# B&R Automation Studio project TrakBasisProject
Automation Studio 6.7.0.187; technology packages: mappCockpit 6.7.0, mappMotion 6.7.2, mappView 6.7.0, OpcUaCs 6.7.0

## Configuration Config1

CPU 5PC900.TS17-00, AutomationRuntime 6.7.8, Build 11.3.0

### Task classes (Cpu.sw)
```
Cyclic#1 (cycle 800 us, tolerance 0 us):
  TrakCtrl <- TrakBasis.TrakCtrl.prg
  utTrakCtrl <- UnitTest.utTrakCtrl.utTrakCtrl.prg
Cyclic#8 (cycle 9600 us):
  TrakHmiCtr <- TrakHmi.TrakHmiCtrl.prg
DataObjects: McAcpSys
NcDataObjects: McDriveLog
Binaries: FWRules, TCData, udbdef, mvLoader, mvConfig, McAcpSim, McAcpDrv, User, iomap, Config_1, arconfig, asfw, ashwac, sysconf, Settings, Role, UaCsConfig, ashwd, Config_3, mCoWebSc, Config_2, BRRole, Hierarchy, TrakHmi
Libraries: runtime, AsZip, FileIO, AsIODiag, AsBrStr, standard, AsARCfg, sys_lib, UnitTest, UtMgr, UtWs, McBase, MpBase, MpAxis, McAcpAx, McAcpTrak, McAxis, CoTrace, arsvcreg, astime, arssl, uacoalprv, powerlnk, AsIecCon, UaCoal, AsEPL, AsIOAcc, AsIoTrc, UaCore, arcoal
```

### Hardware
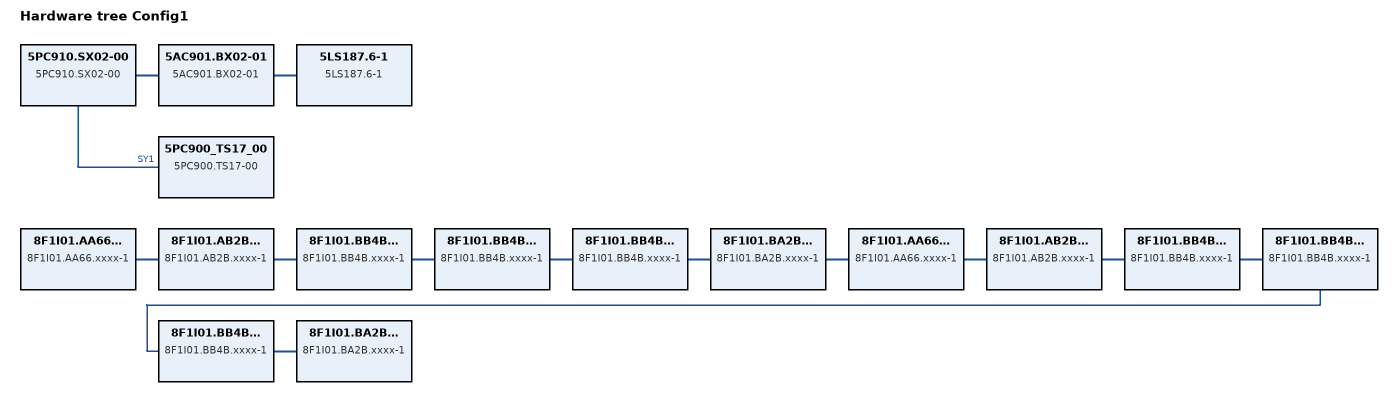
```
5AC901.BX02-01 : 5AC901.BX02-01 v1.1.1.0  [SY -> 5PC910.SX02-00.SY3]
5LS187.6-1 : 5LS187.6-1 v1.10.0.0  [SL -> 5AC901.BX02-01.SL2]
  Connector IF2:
    CycleTime = 800
    EplNatSubnet = 192.168.102.0
5PC900_TS17_00 : 5PC900.TS17-00 v2.2.0.0  [SY -> 5PC910.SX02-00.SY1]
  ConfigurationID = TrakBasisProject_Config1
  UserPartitionSize = 200
  Simulation = 1
  RemMemDevice = PCI.2.LS187.SRAM
  RemMemSize = 20000
  RemanentGlobalPvSize = 3000
  MotionLoggerSize = 2048000
  TimerDeviceType = EPLX2X
  TimerDevice = 5LS187.6-1.IF2
  IdleTaskClass = 3
  TaskClassIdleTime = 1600
  Cyclic1Duration = 800
  Cyclic1Tolerance = 0
  Cyclic1Stack = 256000
  Cyclic1Output = 1
  Cyclic2Duration = 1600
  Cyclic2Tolerance = 1600
  Cyclic3Duration = 20000
  Cyclic3Tolerance = 40000
  Cyclic8Duration = 9600
  Cyclic8Stack = 100000
  FileDevice1
  FileDeviceName1 = SvgData
  FileDevicePath1 = USER_PATH
  ActivateFtpServer = 1
  FtpUser1
  FtpUsername1 = BR
  FtpUserPassword1 = sCAcS4M0KXkF12D2Ev+1iYDIV5DbZPUJhKJtxWH0zr0=  // BR
  FtpUserSalt1 = M7Jis0HY
  FTPAccessRight1 = 0
  FTPdevice1 = ALL
  ActivateWebServer = 1
  WebServerProtocol = 1
  ActivateSdm = 1
5PC910.SX02-00 : 5PC910.SX02-00 v2.1.2.0
  Connector IF1:
    AssignedOperatingSystem = ARemb
  Connector IF3:
    AssignedOperatingSystem = ARemb
    ActivateDevice = 1
  Connector IF4:
    AssignedOperatingSystem = ARemb
    ActivateDevice = 1
    ActivateSnmp = 2
  Connector IF5:
    AssignedOperatingSystem = ARemb
  Connector IF6:
    AssignedOperatingSystem = ARemb
  Connector IF7:
    AssignedOperatingSystem = ARemb
  Connector IF8:
    AssignedOperatingSystem = ARemb
  Connector IF9:
    AssignedOperatingSystem = ARemb
8F1I01.AA66.xxxx-1 : 8F1I01.AA66.xxxx-1 v1.0.1.0 (NodeNumber=12)  [PLK2 -> 8F1I01.AB2B.xxxx-1.PLK1 [Cable Type=PowerlinkCable, Length=10, Version=1.0.0.3]]
  DriveConfiguration:
    McTypeID = LLMConfig
  DriveConfiguration/Segment:
    Shape = STRAIGHT660
    SegmentReference = Seg_7
    SegmentSectorDirection = Positive
  DriveConfiguration/Segment/Compensation:
    ElongationCompensation = UseAssemblySetting
    ACC = Inactive
  DriveConfiguration/Segment:
    StopReaction = UseAssemblySetting
    SpeedFilter = UseAssemblySetting
    PositionControllerLagMonitor = UseAssemblySetting
8F1I01.AA66.xxxx-1a : 8F1I01.AA66.xxxx-1 v1.0.1.0 (NodeNumber=1)  [PLK1 -> 8F1I01.BA2B.xxxx-1a.PLK2 [Cable Type=PowerlinkCable, Length=10, Version=1.0.0.3]; PLK2 -> 8F1I01.AB2B.xxxx-1a.PLK1 [Cable Type=PowerlinkCable, Length=10, Version=1.0.0.3]; PLK3 -> 5LS187.6-1.IF2 [Cable Type=PowerlinkCable, Length=10, Version=1.0.0.3]]
  DriveConfiguration:
    McTypeID = LLMConfig
  DriveConfiguration/Segment:
    Shape = STRAIGHT660
    SegmentReference = Seg_1
    SegmentSectorDirection = Positive
  DriveConfiguration/Segment/Compensation:
    ElongationCompensation = UseAssemblySetting
    ACC = Inactive
  DriveConfiguration/Segment:
    StopReaction = UseAssemblySetting
    SpeedFilter = UseAssemblySetting
    PositionControllerLagMonitor = UseAssemblySetting
8F1I01.AB2B.xxxx-1 : 8F1I01.AB2B.xxxx-1 v1.0.1.0 (NodeNumber=11)  [PLK1 -> 8F1I01.AA66.xxxx-1.PLK2 [Cable Type=PowerlinkCable, Length=10, Version=1.0.0.3]; PLK2 -> 8F1I01.BB4B.xxxx-1c.PLK1 [Cable Type=PowerlinkCable, Length=10, Version=1.0.0.3]]
  DriveConfiguration:
    McTypeID = LLMConfig
  DriveConfiguration/Segment:
    Shape = STRAIGHT105_TO_CIRCULAR
    SegmentReference = Seg_8
    SegmentSectorDirection = Positive
  DriveConfiguration/Segment/Compensation:
    ElongationCompensation = UseAssemblySetting
    ACC = Inactive
  DriveConfiguration/Segment:
    StopReaction = UseAssemblySetting
    SpeedFilter = UseAssemblySetting
    PositionControllerLagMonitor = UseAssemblySetting
8F1I01.AB2B.xxxx-1a : 8F1I01.AB2B.xxxx-1 v1.0.1.0 (NodeNumber=2)  [PLK1 -> 8F1I01.AA66.xxxx-1a.PLK2 [Cable Type=PowerlinkCable, Length=10, Version=1.0.0.3]; PLK2 -> 8F1I01.BB4B.xxxx-1.PLK1 [Cable Type=PowerlinkCable, Length=10, Version=1.0.0.3]]
  DriveConfiguration:
    McTypeID = LLMConfig
  DriveConfiguration/Segment:
    Shape = STRAIGHT105_TO_CIRCULAR
    SegmentReference = Seg_2
    SegmentSectorDirection = Positive
  DriveConfiguration/Segment/Compensation:
    ElongationCompensation = UseAssemblySetting
    ACC = Inactive
  DriveConfiguration/Segment:
    StopReaction = UseAssemblySetting
    SpeedFilter = UseAssemblySetting
    PositionControllerLagMonitor = UseAssemblySetting
8F1I01.BA2B.xxxx-1 : 8F1I01.BA2B.xxxx-1 v1.0.1.0 (NodeNumber=7)  [PLK1 -> 8F1I01.BB4B.xxxx-1b.PLK2 [Cable Type=PowerlinkCable, Length=10, Version=1.0.0.3]]
  DriveConfiguration:
    McTypeID = LLMConfig
  DriveConfiguration/Segment:
    Shape = CIRCULAR_TO_STRAIGHT105
    SegmentReference = Seg_6
    SegmentSectorDirection = Positive
  DriveConfiguration/Segment/Compensation:
    ElongationCompensation = UseAssemblySetting
    ACC = Inactive
  DriveConfiguration/Segment:
    StopReaction = UseAssemblySetting
    SpeedFilter = UseAssemblySetting
    PositionControllerLagMonitor = UseAssemblySetting
8F1I01.BA2B.xxxx-1a : 8F1I01.BA2B.xxxx-1 v1.0.1.0  [PLK1 -> 8F1I01.BB4B.xxxx-1e.PLK2 [Cable Type=PowerlinkCable, Length=10, Version=1.0.0.3]; PLK2 -> 8F1I01.AA66.xxxx-1a.PLK1 [Cable Type=PowerlinkCable, Length=10, Version=1.0.0.3]]
  DriveConfiguration:
    McTypeID = LLMConfig
  DriveConfiguration/Segment:
    Shape = CIRCULAR_TO_STRAIGHT105
    SegmentReference = Seg_12
    SegmentSectorDirection = Positive
  DriveConfiguration/Segment/Compensation:
    ElongationCompensation = UseAssemblySetting
    ACC = Inactive
  DriveConfiguration/Segment:
    StopReaction = UseAssemblySetting
    SpeedFilter = UseAssemblySetting
    PositionControllerLagMonitor = UseAssemblySetting
8F1I01.BB4B.xxxx-1 : 8F1I01.BB4B.xxxx-1 v1.0.1.0 (NodeNumber=4)  [PLK1 -> 8F1I01.AB2B.xxxx-1a.PLK2 [Cable Type=PowerlinkCable, Length=10, Version=1.0.0.3]; PLK2 -> 8F1I01.BB4B.xxxx-1a.PLK1 [Cable Type=PowerlinkCable, Length=10, Version=1.0.0.3]]
  DriveConfiguration:
    McTypeID = LLMConfig
  DriveConfiguration/Segment:
    Shape = CIRCULAR
    SegmentReference = Seg_3
    SegmentSectorDirection = Positive
  DriveConfiguration/Segment/Compensation:
    ElongationCompensation = UseAssemblySetting
    ACC = Inactive
  DriveConfiguration/Segment:
    StopReaction = UseAssemblySetting
    SpeedFilter = UseAssemblySetting
    PositionControllerLagMonitor = UseAssemblySetting
8F1I01.BB4B.xxxx-1a : 8F1I01.BB4B.xxxx-1 v1.0.1.0 (NodeNumber=5)  [PLK1 -> 8F1I01.BB4B.xxxx-1.PLK2 [Cable Type=PowerlinkCable, Length=10, Version=1.0.0.3]; PLK2 -> 8F1I01.BB4B.xxxx-1b.PLK1 [Cable Type=PowerlinkCable, Length=10, Version=1.0.0.3]]
  DriveConfiguration:
    McTypeID = LLMConfig
  DriveConfiguration/Segment:
    Shape = CIRCULAR
    SegmentReference = Seg_4
    SegmentSectorDirection = Positive
  DriveConfiguration/Segment/Compensation:
    ElongationCompensation = UseAssemblySetting
    ACC = Inactive
  DriveConfiguration/Segment:
    StopReaction = UseAssemblySetting
    SpeedFilter = UseAssemblySetting
    PositionControllerLagMonitor = UseAssemblySetting
8F1I01.BB4B.xxxx-1b : 8F1I01.BB4B.xxxx-1 v1.0.1.0 (NodeNumber=6)  [PLK1 -> 8F1I01.BB4B.xxxx-1a.PLK2 [Cable Type=PowerlinkCable, Length=10, Version=1.0.0.3]; PLK2 -> 8F1I01.BA2B.xxxx-1.PLK1 [Cable Type=PowerlinkCable, Length=10, Version=1.0.0.3]]
  DriveConfiguration:
    McTypeID = LLMConfig
  DriveConfiguration/Segment:
    Shape = CIRCULAR
    SegmentReference = Seg_5
    SegmentSectorDirection = Positive
  DriveConfiguration/Segment/Compensation:
    ElongationCompensation = UseAssemblySetting
    ACC = Inactive
  DriveConfiguration/Segment:
    StopReaction = UseAssemblySetting
    SpeedFilter = UseAssemblySetting
    PositionControllerLagMonitor = UseAssemblySetting
8F1I01.BB4B.xxxx-1c : 8F1I01.BB4B.xxxx-1 v1.0.1.0 (NodeNumber=10)  [PLK1 -> 8F1I01.AB2B.xxxx-1.PLK2 [Cable Type=PowerlinkCable, Length=10, Version=1.0.0.3]; PLK2 -> 8F1I01.BB4B.xxxx-1d.PLK1 [Cable Type=PowerlinkCable, Length=10, Version=1.0.0.3]]
  DriveConfiguration:
    McTypeID = LLMConfig
  DriveConfiguration/Segment:
    Shape = CIRCULAR
    SegmentReference = Seg_9
    SegmentSectorDirection = Positive
  DriveConfiguration/Segment/Compensation:
    ElongationCompensation = UseAssemblySetting
    ACC = Inactive
  DriveConfiguration/Segment:
    StopReaction = UseAssemblySetting
    SpeedFilter = UseAssemblySetting
    PositionControllerLagMonitor = UseAssemblySetting
8F1I01.BB4B.xxxx-1d : 8F1I01.BB4B.xxxx-1 v1.0.1.0 (NodeNumber=9)  [PLK1 -> 8F1I01.BB4B.xxxx-1c.PLK2 [Cable Type=PowerlinkCable, Length=10, Version=1.0.0.3]; PLK2 -> 8F1I01.BB4B.xxxx-1e.PLK1 [Cable Type=PowerlinkCable, Length=10, Version=1.0.0.3]]
  DriveConfiguration:
    McTypeID = LLMConfig
  DriveConfiguration/Segment:
    Shape = CIRCULAR
    SegmentReference = Seg_10
    SegmentSectorDirection = Positive
  DriveConfiguration/Segment/Compensation:
    ElongationCompensation = UseAssemblySetting
    ACC = Inactive
  DriveConfiguration/Segment:
    StopReaction = UseAssemblySetting
    SpeedFilter = UseAssemblySetting
    PositionControllerLagMonitor = UseAssemblySetting
8F1I01.BB4B.xxxx-1e : 8F1I01.BB4B.xxxx-1 v1.0.1.0  [PLK1 -> 8F1I01.BB4B.xxxx-1d.PLK2 [Cable Type=PowerlinkCable, Length=10, Version=1.0.0.3]; PLK2 -> 8F1I01.BA2B.xxxx-1a.PLK1 [Cable Type=PowerlinkCable, Length=10, Version=1.0.0.3]]
  DriveConfiguration:
    McTypeID = LLMConfig
  DriveConfiguration/Segment:
    Shape = CIRCULAR
    SegmentReference = Seg_11
    SegmentSectorDirection = Positive
  DriveConfiguration/Segment/Compensation:
    ElongationCompensation = UseAssemblySetting
    ACC = Inactive
  DriveConfiguration/Segment:
    StopReaction = UseAssemblySetting
    SpeedFilter = UseAssemblySetting
    PositionControllerLagMonitor = UseAssemblySetting
```

### Config_1.assembly - 5PC900_TS17_00/mappMotion/Config_1.assembly
```
Element gAssembly_1 (Type=assembly)
  Tracks:
    Track[1]:
      Segments:
        SegmentRef[1] = ::Seg_1
        SegmentRef[2] = ::Seg_2
        SegmentRef[3] = ::Seg_3
        SegmentRef[4] = ::Seg_4
        SegmentRef[5] = ::Seg_5
        SegmentRef[6] = ::Seg_6
        SegmentRef[7] = ::Seg_7
        SegmentRef[8] = ::Seg_8
        SegmentRef[9] = ::Seg_9
        SegmentRef[10] = ::Seg_10
        SegmentRef[11] = ::Seg_11
        SegmentRef[12] = ::Seg_12
  CommonSegmentSettings:
    ControllerParameters:
      DefaultParameter:
        Controller:
          Position:
            ProportionalGain = 150
          Speed:
            ProportionalGain = 120
          FeedForward:
            TotalMass = 1.25
            ForcePositive = 1.0
            ForceNegative = 1.0
  Shuttles:
    MaxShuttleCount = 40
    ShuttleStereotypes:
      ShuttleStRef[1] = ShuttleStereotype_1
    MagnetPlateConfigurations:
      ShuttleType[1] = 8F1Sx.102.xxxxxx-x
    BackupShuttleData = Used
      BackupVar = ::gTrakShBackupRestoreData
```

### Config_2.sector - 5PC900_TS17_00/mappMotion/Config_2.sector
```
Element Sector_1 (Type=sector)
  Type:
    StartSegment:
      SegmentRef = ::Seg_1
    IntermediateSegments:
      SegmentRef[1] = ::Seg_2
      SegmentRef[2] = ::Seg_3
      SegmentRef[3] = ::Seg_4
      SegmentRef[4] = ::Seg_5
      SegmentRef[5] = ::Seg_6
      SegmentRef[6] = ::Seg_7
      SegmentRef[7] = ::Seg_8
      SegmentRef[8] = ::Seg_9
      SegmentRef[9] = ::Seg_10
      SegmentRef[10] = ::Seg_11
    EndSegment:
      SegmentRef = ::Seg_12
      PositionRelativeTo = FromEnd
```

### Config_3.shuttlestereotype - 5PC900_TS17_00/mappMotion/Config_3.shuttlestereotype
```
Element ShuttleStereotype_1 (Type=shuttlestereotype)
  MovementLimits:
    Velocity:
      Velocity = 5.5
    Acceleration:
      Acceleration = 40.0
    Deceleration:
      Deceleration = 40.0
```

### Config_4.assemblyfeature - 5PC900_TS17_00/mappMotion/Config_4.assemblyfeature
```
Element Feature_Shuttle_Auto_Attatch (Type=assemblyfeature)
  Type = ShtSectorAutoAttach
    Priority[1]:
      SectorRef = Sector_1
```

## Logical view

Binary libraries used (declarations not repeated): operator, runtime, AsIecCon, astime, AsZip, FileIO, AsIODiag, AsBrStr, standard, McBase 6.3.0, MpBase 6.7.0, MpAxis 6.3.0, McAcpAx 6.3.0, McAcpTrak 6.7.2, McAxis 6.3.0, CoTrace 6.1.0, UtMgr 6.3.0, sys_lib, AsARCfg, UtWs 6.3.0

### Package Logical/Libraries - Global libraries

### TrakBasis.typ
```iecst
(********************************************************************
 * COPYRIGHT - B&R Spain
 ********************************************************************
 * Package: TrakBasis
 * File: TrakBasis.typ
 * Author: B&R Spain
 * Created: July 22, 2024
 * Modified: July 22, 2024
 ********************************************************************
 * Data types of package TrakBasis for mapp Motion
 ********************************************************************)
(*********************************************************************
* TrakCtrl structures
*********************************************************************)

TYPE
	TrakApplicationErrorEnum :
		(
		TRAK_APP_ERROR_NONE := 0,
		TRAK_APP_ERR_SIM_SH_COUNT_MAX := 100,
		TRAK_APP_ERR_SH_COUNT_MAX := 101,
		TRAK_APP_ERR_SEG_COUNT_MAX := 102,
		TRAK_APP_ERR_SEG_INDEX_MAX := 103,
		TRAK_APP_ERR_NO_SEGMENTS := 104
		);
	TrakCtrlType : 	STRUCT  (*Control structure*)
		Command : TrakCtrlCmdType; (*Command structure*)
		Parameter : TrakCtrlParType; (*Parameter structure*)
		Status : TrakCtrlStatusType; (*Status structure*)
	END_STRUCT;
	TrakCtrlCmdType : 	STRUCT  (*Command structure*)
		Power : BOOL; (*Switch on the controller*)
		Move : TrakCtrlCmdMoveType; (*Movement structures*)
		ErrorReset : BOOL; (*Reset the error in assembly*)
		Recover : TrakCtrlCmdRecoverType; (*Shuttle identity recovery commands*)
	END_STRUCT;
	TrakCtrlCmdMoveType : 	STRUCT  (*Movement structures*)
		Absolute : BOOL; (*Elastic move absolute of all the shuttles to a predefined position*)
		Velocity : BOOL; (*Velocity move of all the shuttles within the predefined sector*)
		Halt : BOOL; (*Stops all shuttle movements*)
	END_STRUCT;
	TrakCtrlCmdRecoverType : 	STRUCT  (*Shuttle identity recovery commands*)
		Index : UINT; (*Index in Status.Shuttle[] of the shuttle to identify*)
		UserID : STRING[32]; (*UserID supplied externally (e.g. by a camera recognition system)*)
		Execute : BOOL; (*Assigns UserID to the shuttle at Index*)
		ResetShuttleData : BOOL; (*Wipes the remanent shuttle backup/restore store (mcACPTRAK_RESTORE_RESET_DATA)*)
	END_STRUCT;
	TrakCtrlParType : 	STRUCT  (*Parameter structure*)
		Position : LREAL; (*Position of the commanded movement for the selecred shuttle*)
		Direction : McDirectionEnum; (*Direction of the commanded movement for the selecred shuttle*)
		Speed : REAL; (*Velocity of the commanded movement for the selecred shuttle*)
		Acceleration : REAL; (*Acceleration of the commanded movement for the selecred shuttle*)
		Deceleration : REAL; (*Deceleration of the commanded movement for the selecred shuttle*)
		RestoreEnabled : BOOL; (*The system try to restore shuttle positions after power on*)
		RestoreTolerance : LREAL; (*Discrepancy allowed when restoring position*)
		SimulationParameters : TrakCtrlParSimType; (*Simulation parameter for the trak system*)
	END_STRUCT;
	TrakCtrlParSimType : 	STRUCT  (*Parameter for when trak is being simulated*)
		Position : LREAL; (*Position of first shuttle*)
		Separation : LREAL; (*Separation between shuttles*)
		Quantity : UINT; (*Quantity of the shuttles*)
	END_STRUCT;
	TrakCtrlStatusType : 	STRUCT  (*Status structure*)
		CommunicationReady : BOOL; (*Communication is posible with the assembly*)
		ReadyForPowerOn : BOOL; (*Assembly can be powered on*)
		PowerOn : BOOL; (*Assembly is powered in*)
		MovementDetected : BOOL; (*There are movements in the assembly*)
		Error : BOOL; (*A hardware or application error is active*)
		ErrorInfo : TrakCtrlStatusErrorInfoType; (*Hardware or application error information*)
		AutomaticRestoreSuccess : BOOL; (*TRUE if the automatic restore matched all detected shuttles; FALSE otherwise (some need Command.Recover)*)
		PLCopenState : TrakCtrlStatusPLCopenStateType; (*PLC Open state of the assembly *)
		Segment : ARRAY[0..TRAK_MAX_SEGMENT_MINUS_ONE]OF TrakCtrlStatusSegmentType; (*Overall count of the segments*)
		Shuttle : ARRAY[0..TRAK_MAX_SHUTTLE_MINUS_ONE]OF TrakCtrlStatusShuttleType; (*Overall count of the shuttles*)
	END_STRUCT;
	TrakCtrlStatusErrorInfoType : 	STRUCT  (*Track error related information*)
		ID : DINT; (*The error id of any ocurred error*)
		Text : STRING[255]; (*Error description*)
		Initiator : STRING[32]; (*Error initiator*)
	END_STRUCT;
	TrakCtrlStatusShuttleType : 	STRUCT  (*Overrall numbers of shuttles*)
		Valid : BOOL; (*Shuttle data valid*)
		Axis : McAxisType; (*McAxis of shuttle*)
		ID : UDINT; (*User defined shuttle ID*)
		Name : STRING[32]; (*User defined name identificator*)
		ActSectorType : McAcpTrakSecTypeEnum; (*Shuttle current sector type*)
		ActSector : STRING[32]; (*Shuttle current sector*)
		ActPosition : LREAL; (*Shuttle position on sector*)
		ActVelocity : REAL; (*Shuttle velocity on sector*)
		TotalMoveDistance : LREAL; (*Shuttle total moved distance*)
		IsConvoyMaster : BOOL; (*Shuttle is a convoy master*)
		Pos : McPosType; (*Shuttle position in the coordinate system*)
		State : TrakCtrlStatusShuttleStateType; (*Shuttle state*)
	END_STRUCT;
	TrakCtrlStatusShuttleStateType : 	STRUCT  (*Shuttle PLCopen state*)
		StatusStandStill : BOOL; (*Shuttle is in state Standstill*)
		StatusStopping : BOOL; (*Shuttle is in state Stopping*)
		StatusErrorStop : BOOL; (*Shuttle is in state Errorstop*)
		StatusDiscreteMotion : BOOL; (*Shuttle is in state DiscreteMotion*)
		StatusContinuousMotion : BOOL; (*Shuttle is in state ContinuousMotion*)
		StatusSynchronizedMotion : BOOL; (*Shuttle is in state SynchronizedMotion*)
	END_STRUCT;
	TrakCtrlStatusPLCopenStateType : 	STRUCT  (*PLC Open states of the assembly*)
		Disabled : BOOL; (*Assembly in disabled state*)
		Homing : BOOL; (*Assembly in homing state*)
		Ready : BOOL; (*Assembly in ready state*)
		Stopping : BOOL; (*Assembly in stopping state*)
		ErrorStop : BOOL; (*Assembly in error state*)
		StartUp : BOOL; (*Assembly in start up state*)
		InvalidConfigurartion : BOOL; (*Assembly is invalid*)
	END_STRUCT;
	TrakCtrlStatusSegmentType : 	STRUCT  (*Overrall numbers of segments*)
		Valid : BOOL; (*Segment data valid*)
		Segment : McSegmentType; (*Segment reference*)
		Name : STRING[32]; (*Segment name (used mainly for diagnostics)*)
		State : TrakCtrlStatusSegmentState; (*Segment current PLCopen state*)
		Info : TrakCtrlStatusSegmentInfoType; (*Segment additional information (tempreature, current...etc)*)
	END_STRUCT;
	TrakCtrlStatusSegmentState : 	STRUCT  (*Segment PLCopen state*)
		StatusDisabled : BOOL; (*Segment is in state Disabled*)
		StatusReady : BOOL; (*Segment is in state Ready*)
		StatusErrorStop : BOOL; (*Segment is in state ErrorStop*)
		InvalidConfig : BOOL; (*Segment has an invalid configuration*)
	END_STRUCT;
	TrakCtrlStatusSegmentInfoType : 	STRUCT  (*Additional segment information*)
		TempBalancer : REAL; (*Internal segment temperature*)
		TempSensor : REAL; (*Backside segment temperature*)
		TempAir : REAL; (*CPU segment temperature*)
		Voltage : REAL; (*DC segment voltage*)
		PowerConsumption : REAL; (*Power consumption of the segment*)
	END_STRUCT;
END_TYPE
```

### TrakBasis.var
```iecst
(**)
(********************************************************************
 * CONSTANT VALUE
********************************************************************)
VAR CONSTANT
	TRAK_MAX_SEGMENT : UINT := 12;
	TRAK_MAX_SHUTTLE : UINT := 40; (*Maximum number of shuttles. This value must match the assembly configuration file*)
	TRAK_MAX_SEGMENT_MINUS_ONE : UINT := TRAK_MAX_SEGMENT-1;
	TRAK_MAX_SHUTTLE_MINUS_ONE : UINT := TRAK_MAX_SHUTTLE-1;
	TRAK_SH_USER_DATA_SIZE : UINT := 0; (*Bytes reserved per shuttle in User data size.This value must match the shuttle stereotype configuration file*)
	// Per B&R docs: array size must be at least MaxShuttleCount * (68 + user data size)
	TRAK_SH_BACKUP_SIZE_MINUS_ONE : UINT := (TRAK_MAX_SHUTTLE*(68+TRAK_SH_USER_DATA_SIZE))-1;
END_VAR
(********************************************************************
 * Global control variable
********************************************************************)
VAR
	gTrakCtrl : TrakCtrlType;
END_VAR
(********************************************************************
 * Backup and restore data - referenced by name from the assembly's
 * "Backup and restore data" configuration element (Config_1.assembly)
********************************************************************)
VAR RETAIN
	gTrakShBackupRestoreData : ARRAY[0..TRAK_SH_BACKUP_SIZE_MINUS_ONE] OF USINT;
END_VAR
```

### Program Logical/TrakBasis/TrakCtrl (IEC)

#### Reference.st
```iecst
(********************************************************************
 * COPYRIGHT - B&R Spain
 ********************************************************************
 * Program: TrakCtrl
 * File: References.st
 * Author: B&R Spain
 * Created: July 22, 2024
 * Modified: July 22, 2024
 ********************************************************************
 * Implementation of program TrakCtrl
 ********************************************************************
 * Gets the references to the structures
 ********************************************************************)
ACTION References:

	// Obtain the address of the global assembly structure. This pointer can be used in other places to read/write the assembly's data.
	AdrAssembly := ADR(gAssembly_1);
	// Obtain the address of the default sector structure where initial shuttle movements will be performed.
	AdrSector := ADR(Sector_1);
	// Store the name of the global assembly for identification or logging purposes.
	AssemblyName := 'gAssembly_1';
	// Access the address of gTrakCtrl using the built-in ACCESS operator. This ensures pTrakCtrl points directly to gTrakCtrl for control operations.
	pTrakCtrl ACCESS ADR(gTrakCtrl);

END_ACTION
```

#### InitSequence.st
```iecst
//********************************************************************
// COPYRIGHT - B&R Spain
//********************************************************************
// Program: TrakCtrl
// File: InitSequence.st
// Author: B&R Spain
// Created: July 22, 2024
//********************************************************************
// Implementation of program TrakCtrl
//********************************************************************
// This action implements a state machine to initialize the AcoposTrak system.
//********************************************************************

ACTION InitSequence:

	// State machine controlling the initialization of the AcoposTrak system
	CASE InitState OF

		INIT_STATE_SET_PARAMETER:

			// Set default motion parameters before communicating with the trak
			pTrakCtrl.Parameter.Speed := 0.5;
			pTrakCtrl.Parameter.Acceleration := 5.0;
			pTrakCtrl.Parameter.Deceleration := 5.0;
			pTrakCtrl.Parameter.Position := 0.0;
			pTrakCtrl.Parameter.Direction := mcDIR_POSITIVE;

			// Additional parameters for simulation and restore operations
			pTrakCtrl.Parameter.SimulationParameters.Position := 0.1;
			pTrakCtrl.Parameter.SimulationParameters.Quantity := 20;
			pTrakCtrl.Parameter.SimulationParameters.Separation := 0.06;
			pTrakCtrl.Parameter.RestoreEnabled := TRUE;
			pTrakCtrl.Parameter.RestoreTolerance := 0.25;

			InitState := INIT_STATE_CHECK_ASM_COMM;

		INIT_STATE_CHECK_ASM_COMM:

			 // Verify that the assembly is ready for communication
			IF (MC_BR_AsmReadInfo_AcpTrak_0.AssemblyInfo.CommunicationReady) THEN
				InitState := INIT_STATE_ASM_RDY_TO_POWER;
			END_IF

		INIT_STATE_ASM_RDY_TO_POWER:

			// Verify that the assembly is ready to be powered on
			IF (MC_BR_AsmReadInfo_AcpTrak_0.AssemblyInfo.ReadyForPowerOn) THEN
				InitState := INIT_STATE_GET_SEGMENT;
			END_IF

		INIT_STATE_GET_SEGMENT:

			// Start retrieving segment information
			MC_BR_AsmGetSegment_AcpTrak_0.Enable := TRUE;
			MC_BR_AsmGetSegment_AcpTrak_0.Next := FALSE;
			Counter := 0;

			InitState := INIT_STATE_GET_SEGMENT_WAIT;

		INIT_STATE_GET_SEGMENT_WAIT:

			IF (MC_BR_AsmGetSegment_AcpTrak_0.Error) THEN
				MC_BR_AsmGetSegment_AcpTrak_0.Enable := FALSE;
				InitState := INIT_STATE_ERROR;

			// If there's no error, check if valid data is available
			ELSIF (MC_BR_AsmGetSegment_AcpTrak_0.Valid) THEN

				// Store the total amount of segments
				TotalCountSegment := MC_BR_AsmGetSegment_AcpTrak_0.TotalCount;

				// An assembly without segments cannot be initialized
				IF (TotalCountSegment = 0) THEN
					MC_BR_AsmGetSegment_AcpTrak_0.Enable := FALSE;
					MC_BR_AsmGetSegment_AcpTrak_0.Next := FALSE;
					pTrakCtrl.Status.Error := TRUE;
					pTrakCtrl.Status.ErrorInfo.ID := TRAK_APP_ERR_NO_SEGMENTS;
					pTrakCtrl.Status.ErrorInfo.Initiator := 'Application';
					pTrakCtrl.Status.ErrorInfo.Text := 'No segments detected in the assembly. Initialization aborted.';
					InitState := INIT_STATE_ERROR;

				// The configured array must be able to hold every detected segment
				ELSIF (TotalCountSegment > TRAK_MAX_SEGMENT) THEN
					MC_BR_AsmGetSegment_AcpTrak_0.Enable := FALSE;
					MC_BR_AsmGetSegment_AcpTrak_0.Next := FALSE;
					pTrakCtrl.Status.Error := TRUE;
					pTrakCtrl.Status.ErrorInfo.ID := TRAK_APP_ERR_SEG_COUNT_MAX;
					pTrakCtrl.Status.ErrorInfo.Initiator := 'Application';
					AuxString := UINT_TO_STRING(TotalCountSegment);
					pTrakCtrl.Status.ErrorInfo.Text := CONCAT('Detected segment count (',AuxString);
					pTrakCtrl.Status.ErrorInfo.Text := CONCAT(pTrakCtrl.Status.ErrorInfo.Text,') exceeds TRAK_MAX_SEGMENT limit (');
					AuxString := UINT_TO_STRING(TRAK_MAX_SEGMENT);
					pTrakCtrl.Status.ErrorInfo.Text := CONCAT(pTrakCtrl.Status.ErrorInfo.Text,AuxString);
					pTrakCtrl.Status.ErrorInfo.Text := CONCAT(pTrakCtrl.Status.ErrorInfo.Text,'). Initialization aborted.');
					InitState := INIT_STATE_ERROR;

				// Protect the destination array if the FB returns inconsistent count information
				ELSIF (Counter >= TRAK_MAX_SEGMENT) THEN
					MC_BR_AsmGetSegment_AcpTrak_0.Enable := FALSE;
					MC_BR_AsmGetSegment_AcpTrak_0.Next := FALSE;
					pTrakCtrl.Status.Error := TRUE;
					pTrakCtrl.Status.ErrorInfo.ID := TRAK_APP_ERR_SEG_INDEX_MAX;
					pTrakCtrl.Status.ErrorInfo.Initiator := 'Application';
					AuxString := UINT_TO_STRING(Counter);
					pTrakCtrl.Status.ErrorInfo.Text := CONCAT('Segment index (',AuxString);
					pTrakCtrl.Status.ErrorInfo.Text := CONCAT(pTrakCtrl.Status.ErrorInfo.Text,') is outside TRAK_MAX_SEGMENT capacity (');
					AuxString := UINT_TO_STRING(TRAK_MAX_SEGMENT);
					pTrakCtrl.Status.ErrorInfo.Text := CONCAT(pTrakCtrl.Status.ErrorInfo.Text,AuxString);
					pTrakCtrl.Status.ErrorInfo.Text := CONCAT(pTrakCtrl.Status.ErrorInfo.Text,'). Initialization aborted.');
					InitState := INIT_STATE_ERROR;

				ELSE

					pTrakCtrl.Status.Segment[Counter].Segment := MC_BR_AsmGetSegment_AcpTrak_0.Segment;

					// Check if all segments are read
					IF (MC_BR_AsmGetSegment_AcpTrak_0.RemainingCount = 0) THEN
						// All segments are retreived -> Move on
						MC_BR_AsmGetSegment_AcpTrak_0.Enable := FALSE;
						MC_BR_AsmGetSegment_AcpTrak_0.Next := FALSE;
						InitState := INIT_STATE_DONE;

					ELSE
						// Still have more segments to retrieve -> Read the next one
						MC_BR_AsmGetSegment_AcpTrak_0.Next := FALSE;
						InitState := INIT_STATE_GET_SEGMENT_NEXT;
					END_IF
				END_IF
			END_IF

		INIT_STATE_GET_SEGMENT_NEXT:

			Counter := Counter + 1;
			MC_BR_AsmGetSegment_AcpTrak_0.Next := TRUE;
			InitState := INIT_STATE_GET_SEGMENT_WAIT;

		INIT_STATE_DONE:

			// Successfully completed the initialization process
			InitDone :=	TRUE;

		INIT_STATE_ERROR:

			// Wait until there are no more active errors. Error handling is managed by TrakCtrl task.
			// After the error has been reset, try again to repeat the initialization sequence.
			IF NOT pTrakCtrl.Status.Error THEN
				InitState := INIT_STATE_CHECK_ASM_COMM;
			END_IF

	END_CASE

END_ACTION
```

#### TrakCtrl.st - Init, cyclic, exit code
```iecst
//*********************************************************************************************************************
// COPYRIGHT - B&R Spain
//*********************************************************************************************************************
// Program: TrakCtrl
// File: TrakCtrl.st
// Author: B&R Spain
// Created: July 22, 2024
//*********************************************************************************************************************
// Implementation of program TrakCtrl
//*********************************************************************************************************************
// Description:
//  - This program initializes and controls the main AcoposTrak assembly.
//  - Handles assembly power states, shuttle management, error handling,
//    and movement commands through a state machine.
//*********************************************************************************************************************

PROGRAM _INIT

	// Initialization of state machines
	InitState := INIT_STATE_SET_PARAMETER;
	TrakState := TRAK_STATE_DISABLED;

	gTrakShBackupRestoreData;

	// Determine if the CPU is running in simulation mode
	InSimulation := DiagCpuIsSimulated();

END_PROGRAM

PROGRAM _CYCLIC

	//*****************************************************************************************************************
    // GETS REFERENCES TO STRUCTURES
    // ATTENTION: This must be the first part in the cyclic PROGRAM
    //*****************************************************************************************************************
	References;

	//*****************************************************************************************************************
	// INITIALIZATION SEQUENCE
	//*****************************************************************************************************************
	InitSequence;

	//*****************************************************************************************************************
	// FBK CALLS for reading status. EXACTLY ONE PER CYCLE
	//*****************************************************************************************************************

	//*********************** MC_BR_ASMREADINFO_ACPTRAK ***************************************************************
	MC_BR_AsmReadInfo_AcpTrak_0.Assembly := AdrAssembly;
	MC_BR_AsmReadInfo_AcpTrak_0.Enable := NOT MC_BR_AsmReadInfo_AcpTrak_0.Error;
	MC_BR_AsmReadInfo_AcpTrak_0();

	//*********************** MC_BR_ASMREADSTATUS_ACPTRAK *************************************************************
	MC_BR_AsmReadStatus_AcpTrak_0.Assembly := AdrAssembly;
	MC_BR_AsmReadStatus_AcpTrak_0.Enable := NOT MC_BR_AsmReadStatus_AcpTrak_0.Error;
	MC_BR_AsmReadStatus_AcpTrak_0();

	//*****************************************************************************************************************
	// CHECK IF SOME TRAK COMPONENT IS IN ERROR
	//*****************************************************************************************************************
	IF MC_BR_AsmReadStatus_AcpTrak_0.AssemblyErrorStop OR (MC_BR_AsmReadInfo_AcpTrak_0.AssemblyInfo.ShuttleCount.InErrorStop > 0)
		OR (MC_BR_AsmReadInfo_AcpTrak_0.AssemblyInfo.SegmentCount.InErrorStop > 0) THEN
		pTrakCtrl.Status.Error := TRUE;
		TrakState := TRAK_STATE_ERROR;
	END_IF

	//*****************************************************************************************************************
	// MAIN SEQUENCE
	//*****************************************************************************************************************

	CASE TrakState OF

		TRAK_STATE_DISABLED:

			// Waits until InitSequence has finished before accepting commands
			IF InitDone THEN
				IF pTrakCtrl.Command.Power THEN
					PowerOn;
					TrakState := TRAK_STATE_SWITCHING_ON;
				END_IF
			END_IF

		TRAK_STATE_SWITCHING_OFF:

			IF MC_BR_AsmPowerOff_AcpTrak_0.Error THEN
				TrakState := TRAK_STATE_ERROR;
			ELSIF MC_BR_AsmPowerOff_AcpTrak_0.Done THEN
				TrakState := TRAK_STATE_DISABLED;
			END_IF

		TRAK_STATE_SWITCHING_ON:

			IF MC_BR_AsmPowerOn_AcpTrak_0.Error THEN
				TrakState := TRAK_STATE_ERROR;
			ELSIF MC_BR_AsmPowerOn_AcpTrak_0.Done THEN
				TrakState := TRAK_STATE_DEL_SHUTTLE;
			END_IF

			IF NOT pTrakCtrl.Command.Power THEN
				PowerOff;
				TrakState := TRAK_STATE_SWITCHING_OFF;
			END_IF

		TRAK_STATE_DEL_SHUTTLE:

			// Clean the array where the shuttles axis are saved
			brsmemset(ADR(pTrakCtrl.Status.Shuttle),0,SIZEOF(pTrakCtrl.Status.Shuttle));
			DeleteShuttles;
			TrakState := TRAK_STATE_DEL_SHUTTLE_WAIT;

		TRAK_STATE_DEL_SHUTTLE_WAIT:

			IF MC_BR_AsmDeleteShuttle_AcpTrak_0.Error THEN
				TrakState := TRAK_STATE_ERROR;
			ELSIF MC_BR_AsmDeleteShuttle_AcpTrak_0.Done THEN
				TrakState := TRAK_STATE_ADD_SHUTTLE_INIT;
			END_IF

		TRAK_STATE_ADD_SHUTTLE_INIT:

			// Only add shuttles when working in simulation
			IF InSimulation THEN
				// Check if requested quantity exceeds maximum allowed
				IF (pTrakCtrl.Parameter.SimulationParameters.Quantity > TRAK_MAX_SHUTTLE) THEN
					// Set application error for user feedback and abort shuttle adding
					pTrakCtrl.Status.Error := TRUE;
					pTrakCtrl.Status.ErrorInfo.ID := TRAK_APP_ERR_SIM_SH_COUNT_MAX;
					pTrakCtrl.Status.ErrorInfo.Initiator := 'Application';
					AuxString := UINT_TO_STRING(pTrakCtrl.Parameter.SimulationParameters.Quantity);
					pTrakCtrl.Status.ErrorInfo.Text := CONCAT('Requested shuttle quantity (',AuxString);
					pTrakCtrl.Status.ErrorInfo.Text := CONCAT(pTrakCtrl.Status.ErrorInfo.Text,') exceeds TRAK_MAX_SHUTTLE limit (');
					AuxString := UINT_TO_STRING(TRAK_MAX_SHUTTLE);
					pTrakCtrl.Status.ErrorInfo.Text := CONCAT(pTrakCtrl.Status.ErrorInfo.Text,AuxString);
					pTrakCtrl.Status.ErrorInfo.Text := CONCAT(pTrakCtrl.Status.ErrorInfo.Text,'). Operation aborted.');
					// Abort shuttle adding and go to error state
					TrakState := TRAK_STATE_ERROR;
				ELSE
					Counter := 0;
					TrakState := TRAK_STATE_ADD_SHUTTLE;
				END_IF
			ELSE
				TrakState := TRAK_STATE_GET_SHUTTLE_INIT;
			END_IF

		TRAK_STATE_ADD_SHUTTLE:

			IF Counter > (pTrakCtrl.Parameter.SimulationParameters.Quantity - 1) THEN
				TrakState := TRAK_STATE_GET_SHUTTLE_INIT;
			ELSE
				AddShuttles;
				Counter := Counter + 1;
				TrakState := TRAK_STATE_ADD_SHUTTLE_WAIT;
			END_IF

		TRAK_STATE_ADD_SHUTTLE_WAIT:

			IF MC_BR_SecAddShuttle_AcpTrak_0.Error THEN
				TrakState := TRAK_STATE_ERROR;
			ELSIF MC_BR_SecAddShuttle_AcpTrak_0.Done THEN
				TrakState := TRAK_STATE_ADD_SHUTTLE;
			END_IF

		TRAK_STATE_GET_SHUTTLE_INIT:

			MC_BR_SecGetShuttle_AcpTrak_0.Enable := TRUE;
			MC_BR_SecGetShuttle_AcpTrak_0.Next := FALSE;

			Counter := 0;
			TrakState := TRAK_STATE_GET_SHUTTLE_WAIT;

		TRAK_STATE_GET_SHUTTLE:

			Counter := Counter + 1;
			MC_BR_SecGetShuttle_AcpTrak_0.Next := TRUE;
			TrakState := TRAK_STATE_GET_SHUTTLE_WAIT;

		TRAK_STATE_GET_SHUTTLE_WAIT:

			IF (MC_BR_SecGetShuttle_AcpTrak_0.Error) THEN
				MC_BR_SecGetShuttle_AcpTrak_0.Enable := FALSE;
				MC_BR_SecGetShuttle_AcpTrak_0.Next := FALSE;
				TrakState := TRAK_STATE_ERROR;
			ELSIF (MC_BR_SecGetShuttle_AcpTrak_0.Valid) THEN
				TotalCountShuttle := MC_BR_SecGetShuttle_AcpTrak_0.TotalCount;

				IF (MC_BR_SecGetShuttle_AcpTrak_0.TotalCount = 0) THEN
					MC_BR_SecGetShuttle_AcpTrak_0.Enable := FALSE;
					TrakState := TRAK_STATE_STANDSTILL;
				ELSE
					// Abort immediately if shuttle count exceeds maximum (safety critical for real hardware)
					IF (TotalCountShuttle > TRAK_MAX_SHUTTLE) THEN
						// Set application error for user feedback and abort operation
						pTrakCtrl.Status.Error := TRUE;
						pTrakCtrl.Status.ErrorInfo.ID := TRAK_APP_ERR_SH_COUNT_MAX;
						pTrakCtrl.Status.ErrorInfo.Initiator := 'Application';
						AuxString := UINT_TO_STRING(TotalCountShuttle);
						pTrakCtrl.Status.ErrorInfo.Text := CONCAT('Detected shuttle count (',AuxString);
						pTrakCtrl.Status.ErrorInfo.Text := CONCAT(pTrakCtrl.Status.ErrorInfo.Text,') exceeds TRAK_MAX_SHUTTLE limit (');
						AuxString := UINT_TO_STRING(TRAK_MAX_SHUTTLE);
						pTrakCtrl.Status.ErrorInfo.Text := CONCAT(pTrakCtrl.Status.ErrorInfo.Text,AuxString);
						pTrakCtrl.Status.ErrorInfo.Text := CONCAT(pTrakCtrl.Status.ErrorInfo.Text,'). Operation aborted for safety.');
						// Abort shuttle detection - could be dangerous to continue with unrecognized shuttles
						MC_BR_SecGetShuttle_AcpTrak_0.Enable := FALSE;
						MC_BR_SecGetShuttle_AcpTrak_0.Next := FALSE;
						TrakState := TRAK_STATE_ERROR;
					ELSE
						// Continue with shuttle processing - all shuttles within limit
						pTrakCtrl.Status.Shuttle[Counter].Axis := MC_BR_SecGetShuttle_AcpTrak_0.Axis;
						pTrakCtrl.Status.Shuttle[Counter].ID := MC_BR_SecGetShuttle_AcpTrak_0.AdditionalInfo.ShuttleID;

						// All shuttles have been retreived -> proceed
						IF (MC_BR_SecGetShuttle_AcpTrak_0.RemainingCount = 0) THEN
							Counter := 0;
							MC_BR_SecGetShuttle_AcpTrak_0.Enable := FALSE;
							TrakState := TRAK_STATE_SH_RESTORE_DATA_INIT;
						ELSE
							MC_BR_SecGetShuttle_AcpTrak_0.Next := FALSE;
							TrakState := TRAK_STATE_GET_SHUTTLE;
						END_IF
					END_IF
				END_IF
			END_IF

		TRAK_STATE_SH_RESTORE_DATA_INIT:

			pTrakCtrl.Status.AutomaticRestoreSuccess := FALSE;

			// Official restore FB matches previously known shuttles by position; an empty UserID attempts to restore all of them at once
			MC_BR_AsmRestoreShData_AcpTrak_0.AdvancedParameters.Tolerance := pTrakCtrl.Parameter.RestoreTolerance;
			// When restore is disabled, wipe the remanent store instead so a future restore never matches stale identities
			IF pTrakCtrl.Parameter.RestoreEnabled THEN
				MC_BR_AsmRestoreShData_AcpTrak_0.AdvancedParameters.Mode := mcACPTRAK_RESTORE_TRY_RESTORING;
			ELSE
				MC_BR_AsmRestoreShData_AcpTrak_0.AdvancedParameters.Mode := mcACPTRAK_RESTORE_RESET_DATA;
			END_IF
			MC_BR_AsmRestoreShData_AcpTrak_0.Execute := TRUE;

			TrakState := TRAK_STATE_SH_RESTORE_DATA_WAIT;

		TRAK_STATE_SH_RESTORE_DATA_WAIT:

			IF MC_BR_AsmRestoreShData_AcpTrak_0.Error THEN
				TrakState := TRAK_STATE_ERROR;
			ELSIF MC_BR_AsmRestoreShData_AcpTrak_0.Done THEN
				// Reset-data outcome carries no restore-status meaning, so AutomaticRestoreSuccess stays FALSE unless a restore was actually attempted
				IF pTrakCtrl.Parameter.RestoreEnabled THEN
					pTrakCtrl.Status.AutomaticRestoreSuccess := (MC_BR_AsmRestoreShData_AcpTrak_0.Info.Status = mcACPTRAK_RESTORE_SUCCESS);
				END_IF
				// Whether shuttles were matched or not, the system is ready to move; unmatched shuttles keep an empty UserID
				// until identified individually through the TrakShIdState sequence below
				TrakState := TRAK_STATE_STANDSTILL;
			END_IF

		TRAK_STATE_STANDSTILL:

			IF NOT pTrakCtrl.Command.Power THEN
				PowerOff;
				TrakState := TRAK_STATE_SWITCHING_OFF;
			ELSIF pTrakCtrl.Command.Move.Halt THEN
				// Shuttles cannot be halted if trak is in standstill
				pTrakCtrl.Command.Move.Halt := FALSE;
			ELSIF pTrakCtrl.Command.Move.Absolute THEN
				pTrakCtrl.Command.Move.Absolute := FALSE;
				Counter := 0;
				TrakState := TRAK_STATE_MOVE_ABS;
			ELSIF pTrakCtrl.Command.Move.Velocity THEN
				pTrakCtrl.Command.Move.Velocity := FALSE;
				Counter := 0;
				TrakState := TRAK_STATE_MOVE_VEL;
			END_IF

		TRAK_STATE_MOVE_ABS:

			IF (Counter > TRAK_MAX_SHUTTLE_MINUS_ONE) THEN
				TrakState := TRAK_STATE_IN_MOTION;
			ELSIF (pTrakCtrl.Status.Shuttle[Counter].Valid) THEN
				MoveAbsolute;
				TrakState := TRAK_STATE_MOVE_ABS_WAIT;
			ELSE
				Counter := Counter + 1;
			END_IF

		TRAK_STATE_MOVE_ABS_WAIT:

			IF MC_BR_ModuloMoveAbs_AcpTrak_0.Error THEN
				TrakState := TRAK_STATE_ERROR;
			ELSE
				Counter := Counter + 1;
				TrakState := TRAK_STATE_MOVE_ABS;
			END_IF

		TRAK_STATE_MOVE_VEL:

			IF (Counter > TRAK_MAX_SHUTTLE_MINUS_ONE) THEN
				TrakState := TRAK_STATE_IN_MOTION;
			ELSIF (pTrakCtrl.Status.Shuttle[Counter].Valid) THEN
				MoveVelocity;
				TrakState := TRAK_STATE_MOVE_VEL_WAIT;
			ELSE
				Counter := Counter + 1;
			END_IF

		TRAK_STATE_MOVE_VEL_WAIT:

			IF MC_BR_ElasticMoveVel_AcpTrak_0.Error THEN
				TrakState := TRAK_STATE_ERROR;
			ELSE
				Counter := Counter + 1;
				TrakState := TRAK_STATE_MOVE_VEL;
			END_IF

		TRAK_STATE_HALTING:

			IF MC_BR_AsmStop_AcpTrak_0.Error THEN
				TrakState := TRAK_STATE_ERROR;
			ELSIF MC_BR_AsmStop_AcpTrak_0.Done THEN
				TrakState := TRAK_STATE_STANDSTILL;
			END_IF

			IF NOT pTrakCtrl.Command.Power THEN
				PowerOff;
				TrakState := TRAK_STATE_SWITCHING_OFF;
			END_IF

		TRAK_STATE_IN_MOTION:

			IF NOT MC_BR_AsmReadInfo_AcpTrak_0.AssemblyInfo.MovementDetected THEN
				TrakState := TRAK_STATE_STANDSTILL;
			END_IF

			IF NOT pTrakCtrl.Command.Power THEN
				PowerOff;
				TrakState := TRAK_STATE_SWITCHING_OFF;
			ELSIF pTrakCtrl.Command.Move.Halt THEN
				pTrakCtrl.Command.Move.Halt := FALSE;
				Halt;
				TrakState := TRAK_STATE_HALTING;
			ELSIF pTrakCtrl.Command.Move.Absolute THEN
				pTrakCtrl.Command.Move.Absolute := FALSE;
				Counter := 0;
				TrakState := TRAK_STATE_MOVE_ABS;
			ELSIF pTrakCtrl.Command.Move.Velocity THEN
				pTrakCtrl.Command.Move.Velocity := FALSE;
				Counter := 0;
				TrakState := TRAK_STATE_MOVE_VEL;
			END_IF

		TRAK_STATE_STOPPING:

			IF MC_BR_AsmStop_AcpTrak_0.Error THEN
				TrakState := TRAK_STATE_ERROR;
			ELSIF MC_BR_AsmStop_AcpTrak_0.Done THEN
				TrakState := TRAK_STATE_STANDSTILL;
			END_IF

			IF NOT pTrakCtrl.Command.Power THEN
				PowerOff;
				TrakState := TRAK_STATE_SWITCHING_OFF;
			END_IF

		TRAK_STATE_ERROR:

			// Reset PowerON command when an error is detected
			pTrakCtrl.Command.Power := FALSE;

			// Deletes the convoy from the convoy master axis before the error is reset
			FOR i:=0 TO TRAK_MAX_SHUTTLE_MINUS_ONE DO
				IF pTrakCtrl.Status.Shuttle[i].IsConvoyMaster THEN
					MC_BR_ConDelete_AcpTrak_0[i].ConvoyMaster := ADR(pTrakCtrl.Status.Shuttle[i].Axis);
					MC_BR_ConDelete_AcpTrak_0[i].Execute := pTrakCtrl.Status.Shuttle[i].State.StatusErrorStop;
				END_IF
			END_FOR

			// Reset errors in assembly (using "ErrorReset command")
			IF pTrakCtrl.Command.ErrorReset THEN
				// Assembly and segment errors can be reset using MC_BR_AsmReset_AcpTrak FB
				IF MC_BR_AsmReadStatus_AcpTrak_0.AssemblyErrorStop OR (MC_BR_AsmReadInfo_AcpTrak_0.AssemblyInfo.SegmentCount.InErrorStop > 0) THEN
					MC_BR_AsmReset_AcpTrak_0.Execute := NOT MC_BR_AsmReset_AcpTrak_0.Error;
				// Shuttle errors can be reset using MC_Reset
				ELSIF (MC_BR_AsmReadInfo_AcpTrak_0.AssemblyInfo.ShuttleCount.InErrorStop > 0) THEN
					FOR i:=0 TO TRAK_MAX_SHUTTLE_MINUS_ONE DO
						MC_Reset_0[i].Axis := ADR(pTrakCtrl.Status.Shuttle[i].Axis);
						MC_Reset_0[i].Execute := pTrakCtrl.Status.Shuttle[i].State.StatusErrorStop;
					END_FOR
				// When there are no more active hardware errors in the system, reset the command and leave error state
				ELSE
					IF pTrakCtrl.Status.PLCopenState.Disabled THEN
						pTrakCtrl.Command.ErrorReset := FALSE;
						ClearError;
						TrakState := TRAK_STATE_DISABLED;
					ELSIF pTrakCtrl.Status.PLCopenState.Ready THEN
						pTrakCtrl.Command.ErrorReset := FALSE;
						ClearError;
						PowerOff;
						TrakState := TRAK_STATE_SWITCHING_OFF;
					END_IF
				END_IF
			END_IF

	END_CASE

	//*****************************************************************************************************************
	// SHUTTLE USERID ASSIGNMENT - Lets the application identify a shuttle by index at any time (e.g. after the
	// automatic restore left it unmatched, or following a camera/barcode read), which internally triggers
	// MC_BR_ShSetUserID_AcpTrak's own restore-by-ID mechanism from the backup store. Also allows wiping the
	// backup store on demand via the same restore FB used at startup.
	//*****************************************************************************************************************

	CASE TrakShIdState OF

		TRAK_SH_ID_STATE_WAIT:

			IF pTrakCtrl.Command.Recover.Execute THEN
				IF (pTrakCtrl.Command.Recover.Index <= TRAK_MAX_SHUTTLE_MINUS_ONE)
					AND pTrakCtrl.Status.Shuttle[pTrakCtrl.Command.Recover.Index].Valid THEN

					ShIdIndex := pTrakCtrl.Command.Recover.Index;
					MC_BR_ShSetUserID_AcpTrak_0.Axis := ADR(pTrakCtrl.Status.Shuttle[ShIdIndex].Axis);
					MC_BR_ShSetUserID_AcpTrak_0.UserID := pTrakCtrl.Command.Recover.UserID;
					MC_BR_ShSetUserID_AcpTrak_0.Execute := TRUE;

					TrakShIdState := TRAK_SH_ID_STATE_ASSIGN_WAIT;
				END_IF

				pTrakCtrl.Command.Recover.Execute := FALSE;
			ELSIF pTrakCtrl.Command.Recover.ResetShuttleData THEN
				MC_BR_AsmRestoreShData_AcpTrak_0.AdvancedParameters.Mode := mcACPTRAK_RESTORE_RESET_DATA;
				MC_BR_AsmRestoreShData_AcpTrak_0.Execute := TRUE;
				pTrakCtrl.Command.Recover.ResetShuttleData := FALSE;

				TrakShIdState := TRAK_SH_ID_STATE_RESET_WAIT;
			END_IF

		TRAK_SH_ID_STATE_ASSIGN_WAIT:

			IF MC_BR_ShSetUserID_AcpTrak_0.Error THEN
				TrakState := TRAK_STATE_ERROR;
				TrakShIdState := TRAK_SH_ID_STATE_WAIT;
			ELSIF MC_BR_ShSetUserID_AcpTrak_0.Done THEN
				TrakShIdState := TRAK_SH_ID_STATE_WAIT;
			END_IF

		TRAK_SH_ID_STATE_RESET_WAIT:

			IF MC_BR_AsmRestoreShData_AcpTrak_0.Error THEN
				TrakState := TRAK_STATE_ERROR;
				TrakShIdState := TRAK_SH_ID_STATE_WAIT;
			ELSIF MC_BR_AsmRestoreShData_AcpTrak_0.Done THEN
				TrakShIdState := TRAK_SH_ID_STATE_WAIT;
			END_IF

	END_CASE

	//*****************************************************************************************************************
	// READ ERRORS FROM TRAK SYSTEM - Based on suggestions from AS Help Guid: 5a0083f9-675b-490c-a00b-1306522f6dd4
	// 1. ***Deviation from regular operation***: Check if there are elements in the Trak in state "ErrorStop"
	// 2. ***Identification of the "Initiator***: Identify the trigger of an error response ("Initiator")
	// 3. ***Collect detailed information***: Read the the error entry in Logger from the "Initiator".
	//*****************************************************************************************************************

	CASE TrakErrorState OF

		TRAK_ERR_STATE_WAIT:

			// When there is some trak element with an active error, find the initiator
			IF MC_BR_AsmReadStatus_AcpTrak_0.AssemblyErrorStop OR (MC_BR_AsmReadInfo_AcpTrak_0.AssemblyInfo.ShuttleCount.InErrorStop > 0)
				OR (MC_BR_AsmReadInfo_AcpTrak_0.AssemblyInfo.SegmentCount.InErrorStop > 0) THEN
				TrakErrorState := TRAK_ERR_STATE_FIND_INIT_ASM;
			END_IF

		TRAK_ERR_STATE_FIND_INIT_ASM:

			// Checks if the assembly is the error initiator
			IF (MC_BR_AsmReadErrorInfo_AcpTrak_0.ErrorInfo.Initiator) THEN
				AdrErrorComponent := AdrAssembly;
				pTrakCtrl.Status.ErrorInfo.Initiator := 'Assembly';
			END_IF

			// Check if initiator has been found
			IF (AdrErrorComponent <> 0) THEN
				TrakErrorState := TRAK_ERR_STATE_COLLECT_LOG;
			ELSE
				TrakErrorState := TRAK_ERR_STATE_FIND_INIT_SEG;
			END_IF

		TRAK_ERR_STATE_FIND_INIT_SEG:

			// Checks if some segment is the error initiator
			FOR i:=0 TO TRAK_MAX_SEGMENT_MINUS_ONE DO
				IF MC_BR_SegReadErrorInfo_AcpTrak_0[i].ErrorInfo.Initiator THEN
					AdrErrorComponent := ADR(gTrakCtrl.Status.Segment[i].Segment);
					pTrakCtrl.Status.ErrorInfo.Initiator := pTrakCtrl.Status.Segment[i].Name;
					EXIT;
				END_IF
			END_FOR

			// Check if initiator has been found
			IF (AdrErrorComponent <> 0) THEN
				TrakErrorState := TRAK_ERR_STATE_COLLECT_LOG;
			ELSE
				TrakErrorState := TRAK_ERR_STATE_FIND_INIT_SH;
			END_IF

		TRAK_ERR_STATE_FIND_INIT_SH:

			// Check if some shuttle is the initiator
			FOR i:=0 TO TRAK_MAX_SHUTTLE_MINUS_ONE DO
				IF MC_BR_ShReadErrorInfo_AcpTrak_0[i].ErrorInfo.Initiator THEN
					AdrErrorComponent := ADR(gTrakCtrl.Status.Shuttle[i].Axis);
					pTrakCtrl.Status.ErrorInfo.Initiator := pTrakCtrl.Status.Shuttle[i].Name;
					EXIT;
				END_IF
			END_FOR

			// Check if initiator has been found
			IF (AdrErrorComponent <> 0) THEN
				TrakErrorState := TRAK_ERR_STATE_COLLECT_LOG;
			ELSE
				pTrakCtrl.Status.ErrorInfo.Text := 'No initiator component found.';
				TrakErrorState := TRAK_ERR_STATE_DONE;
			END_IF

		TRAK_ERR_STATE_COLLECT_LOG:

			MC_BR_ReadErrorText_0.Component := AdrErrorComponent;
			MC_BR_ReadErrorText_0.Enable := (AdrErrorComponent <> 0);
			MC_BR_ReadErrorText_0.ReadNext := TRUE;
			TrakErrorState := TRAK_ERR_STATE_COLLECT_LOG_WAIT;

		TRAK_ERR_STATE_COLLECT_LOG_WAIT:

			IF MC_BR_ReadErrorText_0.ReadDone THEN
				// Important to record the very first triggered error, the rest will not be recorded.
				pTrakCtrl.Status.ErrorInfo.Text := MC_BR_ReadErrorText_0.ErrorRecords.Record[0].Text;
				pTrakCtrl.Status.ErrorInfo.ID := MC_BR_ReadErrorText_0.ErrorRecords.Record[0].EventID;
				TrakErrorState := TRAK_ERR_STATE_DONE;
			ELSIF MC_BR_ReadErrorText_0.Error THEN
				// When FB ouputs an error is because it could not communicate with motion component
				// In that case, mark it as a generic error and output the error ID
				pTrakCtrl.Status.ErrorInfo.Text := 'Unresponsive motion component.';
				pTrakCtrl.Status.ErrorInfo.ID := MC_BR_ReadErrorText_0.ErrorID;
				TrakErrorState := TRAK_ERR_STATE_DONE;
			END_IF

		TRAK_ERR_STATE_DONE:

			// Exit error state when all hardware errors in the trak system have been resolved
			// Only exit if this is a hardware error (not application error)
			IF NOT MC_BR_AsmReadStatus_AcpTrak_0.AssemblyErrorStop AND NOT (MC_BR_AsmReadInfo_AcpTrak_0.AssemblyInfo.ShuttleCount.InErrorStop > 0)
				AND NOT (MC_BR_AsmReadInfo_AcpTrak_0.AssemblyInfo.SegmentCount.InErrorStop > 0) THEN
				AdrErrorComponent := 0;
				MC_BR_ReadErrorText_0.Enable := FALSE;
				MC_BR_ReadErrorText_0.ReadNext := FALSE;
				TrakErrorState := TRAK_ERR_STATE_WAIT;
			END_IF

	END_CASE

	//*****************************************************************************************************************
	// FBK CALLS for TRAK handling. EXACTLY ONE PER CYCLE
	//*****************************************************************************************************************

	//************************* ASSEMBLY ***************************
	MC_BR_AsmPowerOn_AcpTrak_0.Assembly := AdrAssembly;
	MC_BR_AsmPowerOn_AcpTrak_0();
	MC_BR_AsmPowerOn_AcpTrak_0.Execute := FALSE;

	MC_BR_AsmPowerOff_AcpTrak_0.Assembly := AdrAssembly;
	MC_BR_AsmPowerOff_AcpTrak_0();
	MC_BR_AsmPowerOff_AcpTrak_0.Execute := FALSE;

	MC_BR_AsmGetSegment_AcpTrak_0.Assembly := AdrAssembly;
	MC_BR_AsmGetSegment_AcpTrak_0();

	MC_BR_AsmStop_AcpTrak_0.Assembly := AdrAssembly;
	MC_BR_AsmStop_AcpTrak_0();
	MC_BR_AsmStop_AcpTrak_0.Execute := FALSE;

	MC_BR_AsmDeleteShuttle_AcpTrak_0();
	MC_BR_AsmDeleteShuttle_AcpTrak_0.Execute := FALSE;

	MC_BR_AsmReset_AcpTrak_0.Assembly := AdrAssembly;
	MC_BR_AsmReset_AcpTrak_0();
	MC_BR_AsmReset_AcpTrak_0.Execute := FALSE;

	MC_BR_AsmRestoreShData_AcpTrak_0.Assembly := AdrAssembly;
	MC_BR_AsmRestoreShData_AcpTrak_0();
	MC_BR_AsmRestoreShData_AcpTrak_0.Execute := FALSE;

	//************************* SECTOR ***************************
	MC_BR_SecAddShuttle_AcpTrak_0();
	MC_BR_SecAddShuttle_AcpTrak_0.Execute := FALSE;

	MC_BR_SecGetShuttle_AcpTrak_0.Sector := AdrSector;
	MC_BR_SecGetShuttle_AcpTrak_0();

	//************************* SEGMENTS ***************************
	TON_0.IN := NOT TON_0.Q;
	TON_0.PT := T#5s;
	TON_0();

	//************************* SHUTTLES ***************************
	MC_BR_ModuloMoveAbs_AcpTrak_0();
	MC_BR_ModuloMoveAbs_AcpTrak_0.Execute := FALSE;

	MC_BR_ElasticMoveVel_AcpTrak_0();
	MC_BR_ElasticMoveVel_AcpTrak_0.Execute := FALSE;

	FOR i:=0 TO TRAK_MAX_SHUTTLE_MINUS_ONE DO
		MC_Reset_0[i]();
		MC_Reset_0[i].Execute := FALSE;
	END_FOR

	MC_BR_ShSetUserID_AcpTrak_0();
	MC_BR_ShSetUserID_AcpTrak_0.Execute := FALSE;

	FOR i:=0 TO TRAK_MAX_SHUTTLE_MINUS_ONE DO
		MC_BR_ConDelete_AcpTrak_0[i].AdvancedParameters.Mode := mcACPTRAK_CON_DELETE_ANY_CASE;
		MC_BR_ConDelete_AcpTrak_0[i]();
		MC_BR_ConDelete_AcpTrak_0[i].Execute := FALSE;
	END_FOR

	//*****************************************************************************************************************
	// PROVIDES ERROR INFORMATION
	//*****************************************************************************************************************

	//************************* ASSEMBLY ***************************
	MC_BR_AsmReadErrorInfo_AcpTrak_0.Assembly := AdrAssembly;
	MC_BR_AsmReadErrorInfo_AcpTrak_0.Enable := NOT MC_BR_AsmReadErrorInfo_AcpTrak_0.Error;
	MC_BR_AsmReadErrorInfo_AcpTrak_0();

	//************************* SEGMENTS ***************************
	FOR i:=0 TO TRAK_MAX_SEGMENT_MINUS_ONE DO

		MC_BR_SegReadErrorInfo_AcpTrak_0[i].Segment := ADR(pTrakCtrl.Status.Segment[i].Segment);
		MC_BR_SegReadErrorInfo_AcpTrak_0[i].Enable := (pTrakCtrl.Status.Segment[i].Segment.controlif <> 0);
		MC_BR_SegReadErrorInfo_AcpTrak_0[i]();

	END_FOR

	//************************* SHUTTLES ***************************
	FOR i:=0 TO TRAK_MAX_SHUTTLE_MINUS_ONE DO

		MC_BR_ShReadErrorInfo_AcpTrak_0[i].Axis := ADR(pTrakCtrl.Status.Shuttle[i].Axis);
		MC_BR_ShReadErrorInfo_AcpTrak_0[i].Enable := (pTrakCtrl.Status.Shuttle[i].Axis.controlif <> 0);
		MC_BR_ShReadErrorInfo_AcpTrak_0[i]();

	END_FOR

	//************************* GENERIC - READ LOGGER ENTRIES ***************************
	MC_BR_ReadErrorText_0();

	//*****************************************************************************************************************
	// PROVIDES STATUS
	//*****************************************************************************************************************

	//************************* ASSEMBLY ***************************

	pTrakCtrl.Status.CommunicationReady := MC_BR_AsmReadInfo_AcpTrak_0.AssemblyInfo.CommunicationReady;
	pTrakCtrl.Status.ReadyForPowerOn := MC_BR_AsmReadInfo_AcpTrak_0.AssemblyInfo.ReadyForPowerOn;
	pTrakCtrl.Status.PowerOn := MC_BR_AsmReadInfo_AcpTrak_0.AssemblyInfo.PowerOn;
	pTrakCtrl.Status.MovementDetected := MC_BR_AsmReadInfo_AcpTrak_0.AssemblyInfo.MovementDetected;

	pTrakCtrl.Status.PLCopenState.Disabled := MC_BR_AsmReadInfo_AcpTrak_0.AssemblyInfo.PLCopenState = mcACPTRAK_DISABLED;
	pTrakCtrl.Status.PLCopenState.ErrorStop := MC_BR_AsmReadInfo_AcpTrak_0.AssemblyInfo.PLCopenState = mcACPTRAK_ERRORSTOP;
	pTrakCtrl.Status.PLCopenState.Homing := MC_BR_AsmReadInfo_AcpTrak_0.AssemblyInfo.PLCopenState = mcACPTRAK_HOMING;
	pTrakCtrl.Status.PLCopenState.InvalidConfigurartion := MC_BR_AsmReadInfo_AcpTrak_0.AssemblyInfo.PLCopenState = mcACPTRAK_INVALID_CONFIGURATION;
	pTrakCtrl.Status.PLCopenState.Ready := MC_BR_AsmReadInfo_AcpTrak_0.AssemblyInfo.PLCopenState = mcACPTRAK_READY;
	pTrakCtrl.Status.PLCopenState.StartUp := MC_BR_AsmReadInfo_AcpTrak_0.AssemblyInfo.PLCopenState = mcACPTRAK_STARTUP;
	pTrakCtrl.Status.PLCopenState.Stopping := MC_BR_AsmReadInfo_AcpTrak_0.AssemblyInfo.PLCopenState = mcACPTRAK_STOPPING;

	//************************* SEGMENTS ***************************
	FOR i:=0 TO TRAK_MAX_SEGMENT_MINUS_ONE DO

		MC_BR_SegReadStatus_AcpTrak_0[i].Segment := ADR(pTrakCtrl.Status.Segment[i].Segment);
		MC_BR_SegReadStatus_AcpTrak_0[i].Enable := (pTrakCtrl.Status.Segment[i].Segment.controlif <> 0);
		MC_BR_SegReadStatus_AcpTrak_0[i]();

		pTrakCtrl.Status.Segment[i].Valid := (MC_BR_SegReadStatus_AcpTrak_0[i].Valid);

		IF (pTrakCtrl.Status.Segment[i].Valid) THEN
			pTrakCtrl.Status.Segment[i].State.StatusDisabled := MC_BR_SegReadStatus_AcpTrak_0[i].SegmentDisabled;
			pTrakCtrl.Status.Segment[i].State.StatusReady := MC_BR_SegReadStatus_AcpTrak_0[i].SegmentReady;
			pTrakCtrl.Status.Segment[i].State.StatusErrorStop := MC_BR_SegReadStatus_AcpTrak_0[i].SegmentErrorStop;
			pTrakCtrl.Status.Segment[i].State.InvalidConfig := MC_BR_SegReadStatus_AcpTrak_0[i].SegmentInvalidConfig;
		END_IF

		IF MC_BR_SegGetInfo_AcpTrak_0[i].Done THEN
			pTrakCtrl.Status.Segment[i].Name := MC_BR_SegGetInfo_AcpTrak_0[i].SegmentInfo.Name;
		END_IF

		MC_BR_SegGetInfo_AcpTrak_0[i].Segment := ADR(pTrakCtrl.Status.Segment[i].Segment);
		MC_BR_SegGetInfo_AcpTrak_0[i].Execute := (pTrakCtrl.Status.Segment[i].Segment.controlif <> 0) AND TON_0.Q AND pTrakCtrl.Status.PowerOn;
		MC_BR_SegGetInfo_AcpTrak_0[i]();
		MC_BR_SegGetInfo_AcpTrak_0[i].Execute := FALSE;

		// Segments parameters readings
		// 1. Voltage - Should be 58V in opertation
		SegmentProcessParId[0].DataType := mcACPTRAK_SEG_PARTYPE_REAL;
		SegmentProcessParId[0].ParID := 298;
		SegmentProcessParId[0].VariableAddress := ADR(pTrakCtrl.Status.Segment[i].Info.Voltage);
		// 2. Direct Axis Current - Used to find power consumption
		SegmentProcessParId[1].DataType := mcACPTRAK_SEG_PARTYPE_REAL;
		SegmentProcessParId[1].ParID := 218;
		SegmentProcessParId[1].VariableAddress := ADR(SegmentDCurrent[i]);
		// 3. Q-axis Current - Used to find power consumption
		SegmentProcessParId[2].DataType := mcACPTRAK_SEG_PARTYPE_REAL;
		SegmentProcessParId[2].ParID := 213;
		SegmentProcessParId[2].VariableAddress := ADR(SegmentQCurrent[i]);
		// 4. Temperature Balancer - Warning 90�C / Error at 95�C - Internal ambient temperature of segment
		SegmentProcessParId[3].DataType := mcACPTRAK_SEG_PARTYPE_REAL;
		SegmentProcessParId[3].ParID := 63648;
		SegmentProcessParId[3].VariableAddress := ADR(pTrakCtrl.Status.Segment[i].Info.TempBalancer);
		// 5. Temperature Air - Warning 75�C / Error at 80�C - CPU temperature
		SegmentProcessParId[4].DataType := mcACPTRAK_SEG_PARTYPE_REAL;
		SegmentProcessParId[4].ParID := 63647;
		SegmentProcessParId[4].VariableAddress := ADR(pTrakCtrl.Status.Segment[i].Info.TempAir);
		// 6. Tempreature Sensor - Warning 75�C / Error at 80�C - Back side of segment in the center
		SegmentProcessParId[5].DataType := mcACPTRAK_SEG_PARTYPE_REAL;
		SegmentProcessParId[5].ParID := 861;
		SegmentProcessParId[5].VariableAddress := ADR(pTrakCtrl.Status.Segment[i].Info.TempSensor);
		// 7. Power consumption
		pTrakCtrl.Status.Segment[i].Info.PowerConsumption := pTrakCtrl.Status.Segment[i].Info.Voltage * SQRT(SegmentQCurrent[i]**2 + SegmentDCurrent[i]**2);

		MC_BR_SegProcessParID_AcpTrak_0[i].Segment := ADR(pTrakCtrl.Status.Segment[i].Segment);
		MC_BR_SegProcessParID_AcpTrak_0[i].ChannelIndex := 0;
		MC_BR_SegProcessParID_AcpTrak_0[i].DataAddress := ADR(SegmentProcessParId);
		MC_BR_SegProcessParID_AcpTrak_0[i].NumberOfParIDs := 6;
		IF NOT InSimulation THEN
			MC_BR_SegProcessParID_AcpTrak_0[i].Execute := TON_0.Q AND pTrakCtrl.Status.PowerOn;
		END_IF
		MC_BR_SegProcessParID_AcpTrak_0[i]();
		MC_BR_SegProcessParID_AcpTrak_0[i].Execute := FALSE;

	END_FOR

	//************************* SHUTTLES ***************************
	FOR i:=0 TO TRAK_MAX_SHUTTLE_MINUS_ONE DO

		MC_BR_ShReadInfo_AcpTrak_0[i].Axis := ADR(pTrakCtrl.Status.Shuttle[i].Axis);
		MC_BR_ShReadInfo_AcpTrak_0[i].Enable := (pTrakCtrl.Status.Shuttle[i].Axis.controlif <> 0);
		MC_BR_ShReadInfo_AcpTrak_0[i]();

		MC_BR_ShReadFrame_AcpTrak_0[i].Axis := ADR(pTrakCtrl.Status.Shuttle[i].Axis);
		MC_BR_ShReadFrame_AcpTrak_0[i].CoordSystem := mcMCS;
		MC_BR_ShReadFrame_AcpTrak_0[i].Enable := (pTrakCtrl.Status.Shuttle[i].Axis.controlif <> 0);
		MC_BR_ShReadFrame_AcpTrak_0[i]();

		MC_BR_ShReadSectorPos_AcpTrak_0[i].Axis := ADR(pTrakCtrl.Status.Shuttle[i].Axis);
		MC_BR_ShReadSectorPos_AcpTrak_0[i].Sector := AdrSector;
		MC_BR_ShReadSectorPos_AcpTrak_0[i].Enable := (pTrakCtrl.Status.Shuttle[i].Axis.controlif <> 0);
		MC_BR_ShReadSectorPos_AcpTrak_0[i]();

		MC_ReadStatus_0[i].Axis := ADR(pTrakCtrl.Status.Shuttle[i].Axis);
		MC_ReadStatus_0[i].Enable := (pTrakCtrl.Status.Shuttle[i].Axis.controlif <> 0);
		MC_ReadStatus_0[i]();

		pTrakCtrl.Status.Shuttle[i].Valid := (MC_BR_ShReadInfo_AcpTrak_0[i].Valid AND MC_ReadStatus_0[i].Valid);

		IF(pTrakCtrl.Status.Shuttle[i].Valid)THEN
			pTrakCtrl.Status.Shuttle[i].Name := MC_BR_ShReadInfo_AcpTrak_0[i].ShuttleInfo.AdditionalInfo.UserID;
			pTrakCtrl.Status.Shuttle[i].ActSectorType := MC_BR_ShReadInfo_AcpTrak_0[i].ShuttleInfo.CurrentValues.SectorType;
			pTrakCtrl.Status.Shuttle[i].ActSector := MC_BR_ShReadInfo_AcpTrak_0[i].ShuttleInfo.CurrentValues.SectorName;
			// Important to use MC_BR_ShReadSectorPos to get the absolute current position within the predefined sector
			pTrakCtrl.Status.Shuttle[i].ActPosition := MC_BR_ShReadSectorPos_AcpTrak_0[i].Info.Position;
			pTrakCtrl.Status.Shuttle[i].ActVelocity := MC_BR_ShReadInfo_AcpTrak_0[i].ShuttleInfo.CurrentValues.Velocity;
			pTrakCtrl.Status.Shuttle[i].TotalMoveDistance := MC_BR_ShReadInfo_AcpTrak_0[i].ShuttleInfo.LifeCycleInfo.AbsoluteMovementDistance;
			pTrakCtrl.Status.Shuttle[i].IsConvoyMaster := MC_BR_ShReadInfo_AcpTrak_0[i].ShuttleInfo.ConvoyInfo.IsConvoyMaster;
			pTrakCtrl.Status.Shuttle[i].Pos := MC_BR_ShReadFrame_AcpTrak_0[i].Frame.Pos;
			pTrakCtrl.Status.Shuttle[i].State.StatusStandStill := MC_ReadStatus_0[i].StandStill;
			pTrakCtrl.Status.Shuttle[i].State.StatusStopping := MC_ReadStatus_0[i].Stopping;
			pTrakCtrl.Status.Shuttle[i].State.StatusErrorStop := MC_ReadStatus_0[i].ErrorStop;
			pTrakCtrl.Status.Shuttle[i].State.StatusDiscreteMotion := MC_ReadStatus_0[i].DiscreteMotion;
			pTrakCtrl.Status.Shuttle[i].State.StatusContinuousMotion := MC_ReadStatus_0[i].ContinuousMotion;
			pTrakCtrl.Status.Shuttle[i].State.StatusSynchronizedMotion := MC_ReadStatus_0[i].SynchronizedMotion;
		END_IF

	END_FOR

END_PROGRAM

PROGRAM _EXIT

END_PROGRAM
```

#### Commands.st
```iecst
ACTION PowerOn:

	MC_BR_AsmPowerOn_AcpTrak_0.Execute := TRUE;
	MC_BR_AsmPowerOff_AcpTrak_0.Execute := FALSE;

END_ACTION

ACTION PowerOff:

	MC_BR_AsmPowerOn_AcpTrak_0.Execute := FALSE;
	MC_BR_AsmPowerOff_AcpTrak_0.Execute := TRUE;

END_ACTION

ACTION AddShuttles:

	MC_BR_SecAddShuttle_AcpTrak_0.Sector := AdrSector;
	MC_BR_SecAddShuttle_AcpTrak_0.Position := pTrakCtrl.Parameter.SimulationParameters.Position + pTrakCtrl.Parameter.SimulationParameters.Separation * UINT_TO_LREAL(Counter);
	MC_BR_SecAddShuttle_AcpTrak_0.Velocity := 0.0;
	MC_BR_SecAddShuttle_AcpTrak_0.Orientation := mcDIR_POSITIVE;
	MC_BR_SecAddShuttle_AcpTrak_0.Execute := TRUE;

END_ACTION

ACTION DeleteShuttles:

	MC_BR_AsmDeleteShuttle_AcpTrak_0.Assembly := AdrAssembly;
	MC_BR_AsmDeleteShuttle_AcpTrak_0.Command := mcACPTRAK_SH_DELETE_ALL;
	MC_BR_AsmDeleteShuttle_AcpTrak_0.Execute := TRUE;

END_ACTION

ACTION MoveAbsolute:

	MC_BR_ModuloMoveAbs_AcpTrak_0.Axis := ADR(pTrakCtrl.Status.Shuttle[Counter].Axis);
	MC_BR_ModuloMoveAbs_AcpTrak_0.Position := pTrakCtrl.Parameter.Position;
	MC_BR_ModuloMoveAbs_AcpTrak_0.Velocity := pTrakCtrl.Parameter.Speed;
	MC_BR_ModuloMoveAbs_AcpTrak_0.Acceleration := pTrakCtrl.Parameter.Acceleration;
	MC_BR_ModuloMoveAbs_AcpTrak_0.Deceleration := pTrakCtrl.Parameter.Deceleration;
	MC_BR_ModuloMoveAbs_AcpTrak_0.Direction := pTrakCtrl.Parameter.Direction;
	MC_BR_ModuloMoveAbs_AcpTrak_0.Elastic := TRUE;
	MC_BR_ModuloMoveAbs_AcpTrak_0.Execute := TRUE;

END_ACTION

ACTION MoveVelocity:

	MC_BR_ElasticMoveVel_AcpTrak_0.Axis	:= ADR(pTrakCtrl.Status.Shuttle[Counter].Axis);
	MC_BR_ElasticMoveVel_AcpTrak_0.Velocity	:= pTrakCtrl.Parameter.Speed;
	MC_BR_ElasticMoveVel_AcpTrak_0.Acceleration	:= pTrakCtrl.Parameter.Acceleration;
	MC_BR_ElasticMoveVel_AcpTrak_0.Deceleration := pTrakCtrl.Parameter.Deceleration;
	MC_BR_ElasticMoveVel_AcpTrak_0.Direction := pTrakCtrl.Parameter.Direction;
	MC_BR_ElasticMoveVel_AcpTrak_0.Execute := TRUE;

END_ACTION

ACTION Halt:

	MC_BR_AsmStop_AcpTrak_0.Assembly := AdrAssembly;
	MC_BR_AsmStop_AcpTrak_0.AdvancedParameters.Deceleration := pTrakCtrl.Parameter.Deceleration;
	MC_BR_AsmStop_AcpTrak_0.AdvancedParameters.StopMode := mcSTOPMODE_JERK_LIMIT;
	MC_BR_AsmStop_AcpTrak_0.Execute := TRUE;

END_ACTION

ACTION ClearError:

	pTrakCtrl.Status.ErrorInfo.Text := '';
	pTrakCtrl.Status.ErrorInfo.Initiator := '';
	pTrakCtrl.Status.ErrorInfo.ID := 0;
	pTrakCtrl.Status.Error := FALSE;

END_ACTION
```

#### TrakCtrl.typ - Local data types
```iecst
(********************************************************************
 * COPYRIGHT - B&R Spain
 ********************************************************************
 * Program: AsmCtrl
 * File: AsmCtrl.typ
 * Author: B&R Spain
 * Created: July 22, 2024
 * Modified: July 22, 2024
 ********************************************************************
 * Local data types of program TrakCtrl
 ********************************************************************)

TYPE
	TrakStateEnum :
		(
		TRAK_STATE_DISABLED,
		TRAK_STATE_SWITCHING_OFF,
		TRAK_STATE_SWITCHING_ON,
		TRAK_STATE_STANDSTILL,
		TRAK_STATE_DEL_SHUTTLE,
		TRAK_STATE_DEL_SHUTTLE_WAIT,
		TRAK_STATE_ADD_SHUTTLE_INIT,
		TRAK_STATE_ADD_SHUTTLE,
		TRAK_STATE_ADD_SHUTTLE_WAIT,
		TRAK_STATE_GET_SHUTTLE_INIT,
		TRAK_STATE_GET_SHUTTLE,
		TRAK_STATE_GET_SHUTTLE_WAIT,
		TRAK_STATE_SH_RESTORE_DATA_INIT,
		TRAK_STATE_SH_RESTORE_DATA_WAIT,
		TRAK_STATE_MOVE_ABS,
		TRAK_STATE_MOVE_ABS_WAIT,
		TRAK_STATE_MOVE_VEL,
		TRAK_STATE_MOVE_VEL_WAIT,
		TRAK_STATE_IN_MOTION,
		TRAK_STATE_HALTING,
		TRAK_STATE_STOPPING,
		TRAK_STATE_ERROR
		);
	InitStateEnum :
		(
		INIT_STATE_SET_PARAMETER,
		INIT_STATE_CHECK_ASM_COMM,
		INIT_STATE_ASM_RDY_TO_POWER,
		INIT_STATE_GET_SEGMENT,
		INIT_STATE_GET_SEGMENT_WAIT,
		INIT_STATE_GET_SEGMENT_NEXT,
		INIT_STATE_DONE,
		INIT_STATE_ERROR
		);
	TrakErrorStateEnum :
		(
		TRAK_ERR_STATE_WAIT,
		TRAK_ERR_STATE_FIND_INIT_ASM,
		TRAK_ERR_STATE_FIND_INIT_SEG,
		TRAK_ERR_STATE_FIND_INIT_SH,
		TRAK_ERR_STATE_COLLECT_LOG,
		TRAK_ERR_STATE_COLLECT_LOG_WAIT,
		TRAK_ERR_STATE_DONE
		);
	TrakShIdStateEnum :
		(
		TRAK_SH_ID_STATE_WAIT,
		TRAK_SH_ID_STATE_ASSIGN_WAIT,
		TRAK_SH_ID_STATE_RESET_WAIT
		);
END_TYPE
```

#### TrakCtrl.var - Local variables
```iecst
(********************************************************************
 * COPYRIGHT - B&R Spain
 ********************************************************************
 * Program: AsmCtrl
 * File: AsmCtrll.var
 * Author: B&R Spain
 * Created: July 22, 2024
 * Modified: July 22, 2024
 ********************************************************************
 * Local variables of program AsmCtrl
 *******************************************************************
*)
(********************************************************************
 * References
********************************************************************)
VAR
	AdrAssembly : UDINT;
	AssemblyName : STRING[32];
	AdrSector : UDINT;
	pTrakCtrl : REFERENCE TO TrakCtrlType;
END_VAR
(********************************************************************
 * Sequences
********************************************************************)
VAR
	TrakState : TrakStateEnum;
	TrakErrorState : TrakErrorStateEnum;
	TrakShIdState : TrakShIdStateEnum;
	InitState : InitStateEnum;
END_VAR
(********************************************************************
 * Function Blocks
********************************************************************)
(********************************************************************
 * For assembly
********************************************************************)
VAR
	MC_BR_AsmReadInfo_AcpTrak_0 : MC_BR_AsmReadInfo_AcpTrak; (*Reads information of the assembly *)
	MC_BR_AsmReadStatus_AcpTrak_0 : MC_BR_AsmReadStatus_AcpTrak; (*Reads the PLCopen state of the assembly*)
	MC_BR_AsmGetSegment_AcpTrak_0 : MC_BR_AsmGetSegment_AcpTrak; (*Gets all the assembly segments*)
	MC_BR_AsmPowerOff_AcpTrak_0 : MC_BR_AsmPowerOff_AcpTrak; (*Performs a Power OFF of the assembly*)
	MC_BR_AsmPowerOn_AcpTrak_0 : MC_BR_AsmPowerOn_AcpTrak; (*Performs a Power ON of the assembly*)
	MC_BR_AsmReset_AcpTrak_0 : MC_BR_AsmReset_AcpTrak; (*Resets all assembly and segment related errors*)
	MC_BR_AsmStop_AcpTrak_0 : MC_BR_AsmStop_AcpTrak; (*Stops all shuttle movements*)
	MC_BR_AsmDeleteShuttle_AcpTrak_0 : MC_BR_AsmDeleteShuttle_AcpTrak; (*Deletes all shuttles from an assembly (useful in simulation or when shuttle is lost in real system and references needs to be refreshed)*)
	MC_BR_AsmRestoreShData_AcpTrak_0 : MC_BR_AsmRestoreShData_AcpTrak; (*Restores shuttle identity and position from the official remanent store after power loss*)
END_VAR
(********************************************************************
 * For sector
********************************************************************)
VAR
	MC_BR_SecAddShuttle_AcpTrak_0 : MC_BR_SecAddShuttle_AcpTrak; (*Adds a shuttle to a predefined sector*)
	MC_BR_SecGetShuttle_AcpTrak_0 : MC_BR_SecGetShuttle_AcpTrak;
END_VAR
(********************************************************************
 * For shuttles
*******************************************************************)
VAR
	MC_BR_ModuloMoveAbs_AcpTrak_0 : MC_BR_ModuloMoveAbs_AcpTrak; (*Performs an elastic absolute movement within a predefined sector (Modulo is very useful for closed loop assemblies)*)
	MC_BR_ElasticMoveVel_AcpTrak_0 : MC_BR_ElasticMoveVel_AcpTrak; (*Performs an elastic movement within the predefined sector*)
	MC_BR_ShSetUserID_AcpTrak_0 : MC_BR_ShSetUserID_AcpTrak; (*Defines a shuttle user ID that will be later used for identification in case of error*)
	MC_BR_ShReadSectorPos_AcpTrak_0 : ARRAY[0..TRAK_MAX_SHUTTLE_MINUS_ONE] OF MC_BR_ShReadSectorPos_AcpTrak; (*Reads the sector related shuttle position (very useful for closed loop assemblies)*)
	MC_BR_ShReadInfo_AcpTrak_0 : ARRAY[0..TRAK_MAX_SHUTTLE_MINUS_ONE] OF MC_BR_ShReadInfo_AcpTrak; (*Reads some current values of the shuttles such as the current speed, total distance or current sector.*)
	MC_BR_ShReadFrame_AcpTrak_0 : ARRAY[0..TRAK_MAX_SHUTTLE_MINUS_ONE] OF MC_BR_ShReadFrame_AcpTrak; (*Used to read the XYZ position of each shuttle within the environment (may be used for external representation of the system)*)
	MC_BR_ConDelete_AcpTrak_0 : ARRAY[0..TRAK_MAX_SHUTTLE_MINUS_ONE] OF MC_BR_ConDelete_AcpTrak; (*Deletes shuttle convoy (used before error reset of convoy masters)*)
	MC_ReadStatus_0 : ARRAY[0..TRAK_MAX_SHUTTLE_MINUS_ONE] OF MC_ReadStatus; (*Used to read the current PLCopen state of the shuttles*)
	MC_Reset_0 : ARRAY[0..TRAK_MAX_SHUTTLE_MINUS_ONE] OF MC_Reset; (*Reset of the shuttle errors*)
END_VAR
(********************************************************************
 * For segments
*******************************************************************)
VAR
	MC_BR_SegReadStatus_AcpTrak_0 : ARRAY[0..TRAK_MAX_SEGMENT_MINUS_ONE] OF MC_BR_SegReadStatus_AcpTrak; (*Checks segment current PLCopen state*)
	MC_BR_SegProcessParID_AcpTrak_0 : ARRAY[0..TRAK_MAX_SEGMENT_MINUS_ONE] OF MC_BR_SegProcessParID_AcpTrak; (*Used to read different segment ParIDs*)
	MC_BR_SegGetInfo_AcpTrak_0 : ARRAY[0..TRAK_MAX_SEGMENT_MINUS_ONE] OF MC_BR_SegGetInfo_AcpTrak; (*Used to read the name of each segment*)
	TON_0 : TON; (*Timer used to delay the cyclic read of segment ParIDs such as the temperature*)
END_VAR
(********************************************************************
 * For error diagnosis
*******************************************************************)
VAR
	MC_BR_AsmReadErrorInfo_AcpTrak_0 : MC_BR_AsmReadErrorInfo_AcpTrak; (*Reads error related information for the assembly*)
	MC_BR_SegReadErrorInfo_AcpTrak_0 : ARRAY[0..TRAK_MAX_SEGMENT_MINUS_ONE] OF MC_BR_SegReadErrorInfo_AcpTrak; (*Reads error related information for each segment*)
	MC_BR_ShReadErrorInfo_AcpTrak_0 : ARRAY[0..TRAK_MAX_SHUTTLE_MINUS_ONE] OF MC_BR_ShReadErrorInfo_AcpTrak; (*Reads error related information for each shuttle*)
	MC_BR_ReadErrorText_0 : MC_BR_ReadErrorText; (*FB that reads errors from logger*)
END_VAR
(********************************************************************
 * Temp variables
********************************************************************)
VAR
	i : INT; (*Loop index*)
	Counter : UINT; (*Auxiliar variable used to iterate in array positions*)
	ShIdIndex : UINT; (*Shuttle index currently being assigned an externally supplied UserID*)
	InitDone : BOOL; (*Trak initialization process completed*)
	InSimulation : BOOL; (*Trak is in simulation*)
	TotalCountSegment : UINT; (*Used to detect if maximum count of segments is exceeded*)
	TotalCountShuttle : UINT; (*Used to detect if maximum count of shuttles is exceeded*)
	SegmentDCurrent : ARRAY[0..TRAK_MAX_SEGMENT] OF REAL; (*Used to calculate segment power consumption*)
	SegmentQCurrent : ARRAY[0..TRAK_MAX_SEGMENT] OF REAL; (*Used to calculate segment power consumption*)
	AdrErrorComponent : UDINT; (*Reference to motion component to read the logger entry*)
	SegmentProcessParId : ARRAY[0..5] OF McAcpTrakSegProcessParIDType; (*Used to monitor different ParIDs for every segments*)
	AuxString : STRING[32]; (*Auxiliar string used to parse and define shuttle names for ShuttleUser ID*)
END_VAR
```

### Program Logical/TrakHmi/TrakHmiCtrl (IEC)

#### TrakHmi.st - Init, cyclic, exit code
```iecst
(********************************************************************
 * COPYRIGHT - B&R Spain
 ********************************************************************
 * Program: TrakHmi
 * File: TrakHmi.st
 * Author: B&R Spain
 * Created: August 18, 2026
 ********************************************************************
 * Description:
 *  - Drives the diagnostics diagram shown in the "STATUS" Paper widget
 *    (ContentMain.content -> PaperShuttles) from gTrakCtrl.Status.
 *  - Builds the SVG "transform" command string consumed by mapp View, with
 *    ids built from SVG_ID_SYSTEM_PREFIX + SVG_SEG_NAME/SVG_SH_NAME (TrakHmi.var).
 *    Segments (SvgSegment) and shuttles (SvgShuttle) are kept as separate arrays:
 *    segments are always part OF gAssembly_1_Layout.svg (built BY the ACOPOStrak
 *    object hierarchy tool) and never move, so only their fill ever changes;
 *    shuttles don't exist in that file, so their icons are built as SvgContent
 *    and injected via the Paper widget "svgContent" property (ContentMain.binding),
 *    and they also need display/translate/spin, unlike segments.
 *  - Rebuilt at SVG_REFRESH_TIME instead of every PLC cycle: recomputing this ~50-element string on
 *    every fast controller cycle would be wasted CPU with no visible benefit.
 ********************************************************************)

PROGRAM _INIT

	SvgSegIdPrefix := CONCAT(SVG_ID_SYSTEM_PREFIX, SVG_SEG_NAME);
	SvgShIdPrefix := CONCAT(SVG_ID_SYSTEM_PREFIX, SVG_SH_NAME);

	// Segments: SvgSegIdPrefix1..SvgSegIdPrefix<TRAK_MAX_SEGMENT>
	FOR i := 0 TO TRAK_MAX_SEGMENT_MINUS_ONE DO
		SvgNum := i + 1;
		AuxNum := UINT_TO_STRING(SvgNum);
		SvgSegment[i].ID := CONCAT(SvgSegIdPrefix, AuxNum);
	END_FOR

	// Shuttles: SvgShIdPrefix1..SvgShIdPrefix<TRAK_MAX_SHUTTLE>. Ids are always computed (cheap, needed as
	// soon as ShowShuttles turns TRUE); the icons themselves (SvgContent) are only built when ShowShuttles
	// is already TRUE - see CreateSvgContent.
	FOR i := 0 TO TRAK_MAX_SHUTTLE_MINUS_ONE DO
		SvgNum := i + 1;
		AuxNum := UINT_TO_STRING(SvgNum);
		SvgShuttle[i].ID := CONCAT(SvgShIdPrefix, AuxNum);
	END_FOR

	IF ShowShuttles THEN
		CreateSvgContent;
	ELSE
		SvgContent := '';
	END_IF

END_PROGRAM

PROGRAM _CYCLIC

	IF TON_0.Q THEN

		//*************************************************************************************************************
		// SHOW/HIDE SHUTTLES - edge detection is evaluated here; rebuilding happens after shuttle data is refreshed
		//*************************************************************************************************************
		TrigShowShuttlesOn(CLK := ShowShuttles);
		TrigShowShuttlesOff(CLK := ShowShuttles);

		//*************************************************************************************************************
		// SEGMENTS - color only; always part of the project/assembly, so no display/position logic at all
		//*************************************************************************************************************
		FOR i := 0 TO TRAK_MAX_SEGMENT_MINUS_ONE DO
			IF NOT gTrakCtrl.Status.Segment[i].Valid THEN
				SvgSegment[i].Fill := 0;
			ELSIF gTrakCtrl.Status.Segment[i].State.StatusErrorStop THEN
				SvgSegment[i].Fill := 3;
			ELSIF gTrakCtrl.Status.Segment[i].State.StatusReady THEN
				SvgSegment[i].Fill := 1;
			ELSE
				SvgSegment[i].Fill := 0;
			END_IF
		END_FOR

		//*************************************************************************************************************
		// SHUTTLES - color, position and orientation
		//*************************************************************************************************************
		FOR i := 0 TO TRAK_MAX_SHUTTLE_MINUS_ONE DO
			SvgShuttle[i].Visible := gTrakCtrl.Status.Shuttle[i].Valid AND ShowShuttles;
			IF gTrakCtrl.Status.Shuttle[i].Valid THEN
				IF SvgShuttle[i].UserID <> gTrakCtrl.Status.Shuttle[i].Name THEN
					SvgShuttle[i].UserID := gTrakCtrl.Status.Shuttle[i].Name;
					SvgContentDirty := TRUE;
				END_IF
			ELSIF SvgShuttle[i].UserID <> '' THEN
				SvgShuttle[i].UserID := '';
				SvgContentDirty := TRUE;
			END_IF
			SvgShuttle[i].TranslateX := LREAL_TO_REAL(gTrakCtrl.Status.Shuttle[i].Pos.X) / SVG_MM_PER_UNIT;
			SvgShuttle[i].TranslateY := -LREAL_TO_REAL(gTrakCtrl.Status.Shuttle[i].Pos.Y) / SVG_MM_PER_UNIT;

			// Heading from movement direction, not Frame.Orient.Angle1/2/3: those are an ambiguous multi-valued
			// Euler decomposition for this planar system (same physical heading can show up as completely
			// different Angle1/2/3 combinations - see repo memory) and aren't safely combinable by simple math.
			// Below MIN_HEADING_DELTA_SQ the movement is noise, so the last computed heading is kept as-is.
			DeltaX := gTrakCtrl.Status.Shuttle[i].Pos.X - PrevPosX[i];
			DeltaY := gTrakCtrl.Status.Shuttle[i].Pos.Y - PrevPosY[i];
			IF (DeltaX*DeltaX + DeltaY*DeltaY) > MIN_HEADING_DELTA_SQ THEN
				IF DeltaX > 0.0 THEN
					HeadingRad := ATAN(DeltaY/DeltaX);
				ELSIF DeltaX < 0.0 THEN
					IF DeltaY >= 0.0 THEN
						HeadingRad := ATAN(DeltaY/DeltaX) + PI;
					ELSE
						HeadingRad := ATAN(DeltaY/DeltaX) - PI;
					END_IF
				ELSIF DeltaY > 0.0 THEN
					HeadingRad := PI/2.0;
				ELSE
					HeadingRad := -PI/2.0;
				END_IF
				// SVG y-axis points down (opposite of the real-world coordinate system) - negate to compensate
				SvgShuttle[i].Angle := -LREAL_TO_REAL(HeadingRad * RAD_TO_DEG);
			END_IF
			PrevPosX[i] := gTrakCtrl.Status.Shuttle[i].Pos.X;
			PrevPosY[i] := gTrakCtrl.Status.Shuttle[i].Pos.Y;

			IF NOT gTrakCtrl.Status.PowerOn THEN
				SvgShuttle[i].Fill := 0;
			ELSIF gTrakCtrl.Status.Shuttle[i].State.StatusErrorStop THEN
				SvgShuttle[i].Fill := 3;
			ELSIF gTrakCtrl.Status.Shuttle[i].State.StatusStopping THEN
				SvgShuttle[i].Fill := 2;
			ELSE
				SvgShuttle[i].Fill := 1;
			END_IF
		END_FOR

		//*************************************************************************************************************
		// SVG CONTENT - rebuild only when shown or when a UserID changes (for example after shuttle recovery)
		//*************************************************************************************************************
		IF TrigShowShuttlesOff.Q THEN
			SvgContent := '';
		ELSIF ShowShuttles AND (TrigShowShuttlesOn.Q OR SvgContentDirty) THEN
			CreateSvgContent;
			SvgContentDirty := FALSE;
		END_IF

		//*************************************************************************************************************
		// BUILD THE TRANSFORM STRING - one "select" command per element, in the format expected by widget Paper
		//*************************************************************************************************************
		CreateSvgTransform;

		TON_0.IN := FALSE;
	ELSE
		TON_0.IN := TRUE;
	END_IF

	TON_0.PT := SVG_REFRESH_TIME;
	TON_0();

END_PROGRAM

PROGRAM _EXIT

END_PROGRAM
```

#### TrakHmi.typ - Local data types
```iecst
(********************************************************************
 * COPYRIGHT - B&R Spain
 ********************************************************************
 * Program: TrakHmi
 * File: TrakHmi.typ
 * Author: B&R Spain
 * Created: August 18, 2026
 ********************************************************************
 * Local data types of program TrakHmi
 ********************************************************************)

TYPE
	SvgSegmentType : 	STRUCT  (*Runtime state of one segment - always part of gAssembly_1_Layout.svg, never moves, only its fill changes*)
		ID : STRING[10]; (*<g> id in gAssembly_1_Layout.svg (e.g. gsg_Seg_1)*)
		Fill : UINT; (*Index into the Paper widget colorList (0 Disabled, 1 Ready, 2 Stopping, 3 ErrorStop)*)
	END_STRUCT;
	SvgShuttleType : 	STRUCT  (*Runtime state of one shuttle - shown/hidden, moved, rotated and colored*)
		ID : STRING[10]; (*<g> id built in SvgContent (e.g. gsg_Sh_1)*)
		UserID : STRING[32]; (*UserID displayed next to the shuttle; empty means the shuttle is not identified*)
		Visible : BOOL; (*Element is shown on the diagram*)
		TranslateX : REAL; (*Pixel offset in x-direction*)
		TranslateY : REAL; (*Pixel offset in y-direction*)
		Angle : REAL; (*Rotation in degrees around the element's own origin*)
		Fill : UINT; (*Index into the Paper widget colorList (0 Disabled, 1 Ready, 2 Stopping, 3 ErrorStop)*)
	END_STRUCT;
END_TYPE
```

#### TrakHmi.var - Local variables
```iecst
(********************************************************************
 * COPYRIGHT - B&R Spain
 ********************************************************************
 * Program: TrakHmi
 * File: TrakHmi.var
 * Author: B&R Spain
 * Created: August 18, 2026
 ********************************************************************
 * Local variables of program TrakHmi
 ********************************************************************)
(********************************************************************
 * CONSTANT VALUES
 ********************************************************************)
VAR CONSTANT
	SVG_MM_PER_UNIT : REAL := 1000.0; (*Shuttle.Pos is in mm; gAssembly_1_Layout.svg's viewBox is in m - divide by this to convert*)
	SVG_REFRESH_TIME : TIME := T#50ms; (*Diagram refresh period - also the sampling interval used for the heading-from-movement delta*)
	SVG_ID_SYSTEM_PREFIX : STRING[10] := 'gsg_'; (*Fixed prefix the SVG configuration tool always adds to element ids, regardless of the configured name*)
	SVG_FILL_PREFIX : STRING[4] := 'p'; (*Prefix on the id of whichever element actually carries the fill color - the object hierarchy tool adds it to each segment's nested polygon, and CreateSvgContent adds it to each shuttle's polygon too, since the wrapping <g>'s own fill can never override a child's own fill attribute*)
	SVG_SEG_NAME : STRING[16] := 'Seg_'; (*Configured name for segment elements - only this (and SVG_SH_NAME) should need changing if TrakLayout.svg is renamed*)
	SVG_SH_NAME : STRING[16] := 'Sh_'; (*Configured name for shuttle elements*)
	SVG_CONTENT_VIEWBOX : STRING[40] := '-1.39558 -0.765 2.13115 0.88'; (*Must match gAssembly_1_Layout.svg's own viewBox (its 1st line) - update by hand if the assembly layout changes*)
	PI : LREAL := 3.14159265358979323846;
	RAD_TO_DEG : LREAL := 180.0/PI;
	MIN_HEADING_DELTA_SQ : LREAL := 4.0; (*mm^2 (~2mm move) - below this, movement is noise and the shuttle's heading is left unchanged*)
END_VAR
(********************************************************************
 * Diagram elements
 ********************************************************************)
VAR
	SvgSegment : ARRAY[0..TRAK_MAX_SEGMENT_MINUS_ONE] OF SvgSegmentType;
	SvgShuttle : ARRAY[0..TRAK_MAX_SHUTTLE_MINUS_ONE] OF SvgShuttleType;
	SvgTransform : STRING[8000]; (*Bound to the Paper widget "transform" property (ContentMain.binding)*)
	SvgContent : STRING[24000]; (*Shuttle icons and UserID labels, bound to the Paper widget "svgContent" property; empty whenever ShowShuttles is FALSE*)
	SvgSegIdPrefix : STRING[26]; (*SVG_ID_SYSTEM_PREFIX + SVG_SEG_NAME, computed once in _INIT*)
	SvgShIdPrefix : STRING[26]; (*SVG_ID_SYSTEM_PREFIX + SVG_SH_NAME, computed once in _INIT*)
	PrevPosX : ARRAY[0..TRAK_MAX_SHUTTLE_MINUS_ONE] OF LREAL; (*Shuttle.Pos.X from the previous refresh, used to derive heading from movement direction*)
	PrevPosY : ARRAY[0..TRAK_MAX_SHUTTLE_MINUS_ONE] OF LREAL; (*Shuttle.Pos.Y from the previous refresh, used to derive heading from movement direction*)
	ShowShuttles : BOOL := TRUE; (*Bindable from mapp View (ShowShuttlesButton) - lets the operator hide all shuttles when only segment states matter*)
END_VAR
(********************************************************************
 * Sequence control
 ********************************************************************)
VAR
	i : UINT;
	SvgNum : UINT; (*1-based element number used to build ids SvgSegIdPrefix<n>/SvgShIdPrefix<n> - UINT_TO_STRING requires a plain variable, not an inline expression*)
	AuxNum : STRING[24]; (*Scratch buffer for brsftoa/brsitoa numeric-to-string conversions before appending to SvgTransform via brsstrcat*)
	AuxID : STRING[14]; (*Scratch buffer for an element's fill-select id (SVG_FILL_PREFIX+ID), computed on the fly in CreateSvgTransform*)
	SvgContentDirty : BOOL; (*Requests one SvgContent rebuild after a shuttle UserID changes*)
	XmlUserID : STRING[160]; (*Escaped UserID; worst case is 32 ampersands expanded to &amp;*)
	XmlChar : STRING[1]; (*Single UserID character being escaped for insertion into SVG text*)
	XmlCharCount : INT;
	XmlCharIndex : INT;
	DeltaX : LREAL; (*Pos.X - PrevPosX, scratch for heading-from-movement calculation*)
	DeltaY : LREAL; (*Pos.Y - PrevPosY, scratch for heading-from-movement calculation*)
	HeadingRad : LREAL; (*ATAN2(DeltaY,DeltaX) equivalent, radians, scratch for heading-from-movement calculation*)
	TrigShowShuttlesOn : R_TRIG; (*Rebuilds SvgContent once, on the rising edge of ShowShuttles*)
	TrigShowShuttlesOff : F_TRIG; (*Clears SvgContent once, on the falling edge of ShowShuttles*)
	TON_0 : TON; (*Throttles the diagram rebuild to SVG_REFRESH_TIME instead of every PLC cycle*)
END_VAR
```

#### CreateSvgTransform.st - Builds the SvgTransform command string
```iecst
ACTION CreateSvgTransform:

	//*************************************************************************************************************
	// BUILD THE TRANSFORM STRING - one "select" command per element, in the format expected by widget Paper
	// Built with brsstrcat (not CONCAT: its result is hard-capped at STRING[255], which silently truncated
	// the front of SvgTransform - i.e. dropped earlier segments - once the string grew past that size)
	//*************************************************************************************************************
	SvgTransform := '[';

	//*************************************************************************************************************
	// SEGMENTS - fill only, always emitted (they're always part of the project/assembly). Selects
	// SVG_FILL_PREFIX+ID (the polygon nested inside each gsg_Seg_N group), not ID itself: ID is the
	// <g> wrapper, whose own fill can never override the inline style already set on its child polygon.
	//*************************************************************************************************************
	FOR i := 0 TO TRAK_MAX_SEGMENT_MINUS_ONE DO
		AuxID := CONCAT(SVG_FILL_PREFIX, SvgSegment[i].ID);
		brsstrcat(ADR(SvgTransform), ADR('{"select":"#'));
		brsstrcat(ADR(SvgTransform), ADR(AuxID));
		brsstrcat(ADR(SvgTransform), ADR('","fill":'));
		brsitoa(SvgSegment[i].Fill, ADR(AuxNum));
		brsstrcat(ADR(SvgTransform), ADR(AuxNum));
		brsstrcat(ADR(SvgTransform), ADR('},'));
	END_FOR

	//*************************************************************************************************************
	// SHUTTLES - display, position, orientation and fill. Skipped entirely (not just hidden) while
	// ShowShuttles is FALSE - their icons don't even exist in SvgContent then.
	//*************************************************************************************************************
	IF ShowShuttles THEN
		FOR i := 0 TO TRAK_MAX_SHUTTLE_MINUS_ONE DO
			brsstrcat(ADR(SvgTransform), ADR('{"select":"#'));
			brsstrcat(ADR(SvgTransform), ADR(SvgShuttle[i].ID));
			brsstrcat(ADR(SvgTransform), ADR('","display":'));
			IF NOT SvgShuttle[i].Visible THEN
				brsstrcat(ADR(SvgTransform), ADR('false},'));
			ELSE
				brsstrcat(ADR(SvgTransform), ADR('true'));
				IF (SvgShuttle[i].TranslateX <> 0) OR (SvgShuttle[i].TranslateY <> 0) THEN
					brsstrcat(ADR(SvgTransform), ADR(',"translate":['));
					brsftoa(SvgShuttle[i].TranslateX, ADR(AuxNum));
					brsstrcat(ADR(SvgTransform), ADR(AuxNum));
					brsstrcat(ADR(SvgTransform), ADR(','));
					brsftoa(SvgShuttle[i].TranslateY, ADR(AuxNum));
					brsstrcat(ADR(SvgTransform), ADR(AuxNum));
					brsstrcat(ADR(SvgTransform), ADR(']'));
				END_IF
				brsstrcat(ADR(SvgTransform), ADR('},'));

				// spin/fill go on the inner polygon (AuxID), not the outer <g> (ID): the outer <g> already got
				// translated above, so spinning IT around (0,0) would orbit it around the SVG's global origin
				// instead of its own center - see repo memory for the full reasoning
				AuxID := CONCAT(SVG_FILL_PREFIX, SvgShuttle[i].ID);
				brsstrcat(ADR(SvgTransform), ADR('{"select":"#'));
				brsstrcat(ADR(SvgTransform), ADR(AuxID));
				brsstrcat(ADR(SvgTransform), ADR('","fill":'));
				brsitoa(SvgShuttle[i].Fill, ADR(AuxNum));
				brsstrcat(ADR(SvgTransform), ADR(AuxNum));
				IF SvgShuttle[i].Angle <> 0 THEN
					brsstrcat(ADR(SvgTransform), ADR(',"spin":['));
					brsftoa(SvgShuttle[i].Angle, ADR(AuxNum));
					brsstrcat(ADR(SvgTransform), ADR(AuxNum));
					brsstrcat(ADR(SvgTransform), ADR(',0,0]'));
				END_IF
				brsstrcat(ADR(SvgTransform), ADR('},'));
			END_IF
		END_FOR
	END_IF

	brsstrcat(ADR(SvgTransform), ADR('{}]'));

END_ACTION
```

#### CreateSvgContent.st - Builds the SvgContent string (shuttle icons)
```iecst
ACTION CreateSvgContent:

	//*************************************************************************************************************
	// BUILD SVGCONTENT - shuttle icons and UserID labels only exist here (not in gAssembly_1_Layout.svg). Only called while
	// ShowShuttles is TRUE; the caller clears SvgContent to '' directly when ShowShuttles goes FALSE.
	// Must be wrapped in its own <svg viewBox=...> (matching gAssembly_1_Layout.svg) - without it mapp View
	// does not mount/render the appended elements at all.
	//*************************************************************************************************************
	SvgContent := '<svg version="1.1" xmlns="http://www.w3.org/2000/svg" viewBox="';
	brsstrcat(ADR(SvgContent), ADR(SVG_CONTENT_VIEWBOX));
	brsstrcat(ADR(SvgContent), ADR('">'));
	FOR i := 0 TO TRAK_MAX_SHUTTLE_MINUS_ONE DO
		AuxID := CONCAT(SVG_FILL_PREFIX, SvgShuttle[i].ID);
		brsstrcat(ADR(SvgContent), ADR('<g id="'));
		brsstrcat(ADR(SvgContent), ADR(SvgShuttle[i].ID));
		brsstrcat(ADR(SvgContent), ADR('"><polygon id="'));
		brsstrcat(ADR(SvgContent), ADR(AuxID));
		brsstrcat(ADR(SvgContent), ADR('" points="-0.025,-0.023 0.0125,-0.023 0.025,0 0.0125,0.023 -0.025,0.023 -0.025,-0.023" stroke="black" fill="lightgrey" style="stroke-width:0.004"/>'));

		IF SvgShuttle[i].UserID <> '' THEN
			// The label is a sibling of the rotating polygon. The outer group translates both elements, while
			// CreateSvgTransform spins only the polygon, so the UserID remains horizontal as the shuttle turns.
			// Alternate labels above and below neighboring shuttles to reduce text overlap.
			IF (i MOD 2) = 0 THEN
				brsstrcat(ADR(SvgContent), ADR('<line x1="0" y1="0" x2="0.03" y2="-0.035" stroke="black" stroke-width="0.002"/><text x="0.035" y="-0.04" font-size="0.035" style="fill:black">'));
			ELSE
				brsstrcat(ADR(SvgContent), ADR('<line x1="0" y1="0" x2="0.03" y2="0.035" stroke="black" stroke-width="0.002"/><text x="0.035" y="0.06" font-size="0.035" style="fill:black">'));
			END_IF
			XmlUserID := '';
			XmlCharCount := LEN(SvgShuttle[i].UserID);
			FOR XmlCharIndex := 1 TO XmlCharCount DO
				XmlChar := MID(SvgShuttle[i].UserID, 1, XmlCharIndex);
				IF XmlChar = '&' THEN
					brsstrcat(ADR(XmlUserID), ADR('&amp;'));
				ELSIF XmlChar = '<' THEN
					brsstrcat(ADR(XmlUserID), ADR('&lt;'));
				ELSIF XmlChar = '>' THEN
					brsstrcat(ADR(XmlUserID), ADR('&gt;'));
				ELSE
					brsstrcat(ADR(XmlUserID), ADR(XmlChar));
				END_IF
			END_FOR
			brsstrcat(ADR(SvgContent), ADR(XmlUserID));
			brsstrcat(ADR(SvgContent), ADR('</text>'));
		END_IF
		brsstrcat(ADR(SvgContent), ADR('</g>'));
	END_FOR
	brsstrcat(ADR(SvgContent), ADR('</svg>'));

END_ACTION
```

### Package Logical/UnitTest/utTrakCtrl - Easy mode: focus on writing tests

### Program Logical/UnitTest/utTrakCtrl/utTrakCtrl (ANSIC) - Empty template for use with helper tool

#### variables.var - Name the suite and add PVs for the program
```iecst
(********************************************************************
 * COPYRIGHT --
 ********************************************************************
 * Program: utTemplate_automated
 * File: variables.var
 * Author: -
 * Created: -
 ********************************************************************
 * Local variables of program utTemplate_automated
 ********************************************************************)
(*Describe the test*)
VAR
	Testsuite : UtMgrTestSuite := (Name:='utTrakCtrl',Description:='TrakCtrl unit tests',Type:=utMgrTEST_TYPE_C);
END_VAR
(*Variables used in the tests*)
```

#### autoGeneratedFile.c - Auto generated code - list of all test sets in the program
```c
/*
B+R UnitTest: This is generated code.
Do not edit! Do not move!
Description: UnitTest Testprogramm infrastructure (List of TestSets).
LastUpdated: 2025-09-17 08:43:00Z
By B+R UnitTest Helper Version: 2.0.0.0
*/
#include "UnitTest.h"

UNITTEST_TESTSET_DECLARATION  Set_Testcases;

UNITTEST_TESTSET_FIXTURES(utTestSets)
{
	new_TestSet(Set_Testcases),
};
UNTITTEST_TESTSET_HANDLER();
```
